   STATUS[967].EXT.AlarmPresent := FALSE;
   STATUS[967].EXT.AlarmFailUnAck := FALSE;
   STATUS[967].Status := 0;
   STATUS[967].TimeStamp := 16#0000;
   STATUS[968].EXT.AlarmWarnUnAck := FALSE;
   STATUS[968].EXT.AckRequired := FALSE;
   STATUS[968].EXT.Maintanence := FALSE;
   STATUS[968].EXT.Operation := FALSE;
   STATUS[968].EXT.Forced := FALSE;
   STATUS[968].EXT.BIT29 := FALSE;
   STATUS[968].EXT.BIT30 := FALSE;
   STATUS[968].EXT.BIT31 := FALSE;
   STATUS[968].EXT.ModeBit1 := FALSE;
   STATUS[968].EXT.ModeBit2 := FALSE;
   STATUS[968].EXT.ModeBit3 := FALSE;
   STATUS[968].EXT.BIT19 := FALSE;
   STATUS[968].EXT.BIT20 := FALSE;
   STATUS[968].EXT.AlarmSuppressed := FALSE;
   STATUS[968].EXT.AlarmPresent := FALSE;
   STATUS[968].EXT.AlarmFailUnAck := FALSE;
   STATUS[968].Status := 0;
   STATUS[968].TimeStamp := 16#0000;
   STATUS[969].EXT.AlarmWarnUnAck := FALSE;
   STATUS[969].EXT.AckRequired := FALSE;
   STATUS[969].EXT.Maintanence := FALSE;
   STATUS[969].EXT.Operation := FALSE;
   STATUS[969].EXT.Forced := FALSE;
   STATUS[969].EXT.BIT29 := FALSE;
   STATUS[969].EXT.BIT30 := FALSE;
   STATUS[969].EXT.BIT31 := FALSE;
   STATUS[969].EXT.ModeBit1 := FALSE;
   STATUS[969].EXT.ModeBit2 := FALSE;
   STATUS[969].EXT.ModeBit3 := FALSE;
   STATUS[969].EXT.BIT19 := FALSE;
   STATUS[969].EXT.BIT20 := FALSE;
   STATUS[969].EXT.AlarmSuppressed := FALSE;
   STATUS[969].EXT.AlarmPresent := FALSE;
   STATUS[969].EXT.AlarmFailUnAck := FALSE;
   STATUS[969].Status := 0;
   STATUS[969].TimeStamp := 16#0000;
   STATUS[970].EXT.AlarmWarnUnAck := FALSE;
   STATUS[970].EXT.AckRequired := FALSE;
   STATUS[970].EXT.Maintanence := FALSE;
   STATUS[970].EXT.Operation := FALSE;
   STATUS[970].EXT.Forced := FALSE;
   STATUS[970].EXT.BIT29 := FALSE;
   STATUS[970].EXT.BIT30 := FALSE;
   STATUS[970].EXT.BIT31 := FALSE;
   STATUS[970].EXT.ModeBit1 := FALSE;
   STATUS[970].EXT.ModeBit2 := FALSE;
   STATUS[970].EXT.ModeBit3 := FALSE;
   STATUS[970].EXT.BIT19 := FALSE;
   STATUS[970].EXT.BIT20 := FALSE;
   STATUS[970].EXT.AlarmSuppressed := FALSE;
   STATUS[970].EXT.AlarmPresent := FALSE;
   STATUS[970].EXT.AlarmFailUnAck := FALSE;
   STATUS[970].Status := 0;
   STATUS[970].TimeStamp := 16#0000;
   STATUS[971].EXT.AlarmWarnUnAck := FALSE;
   STATUS[971].EXT.AckRequired := FALSE;
   STATUS[971].EXT.Maintanence := FALSE;
   STATUS[971].EXT.Operation := FALSE;
   STATUS[971].EXT.Forced := FALSE;
   STATUS[971].EXT.BIT29 := FALSE;
   STATUS[971].EXT.BIT30 := FALSE;
   STATUS[971].EXT.BIT31 := FALSE;
   STATUS[971].EXT.ModeBit1 := FALSE;
   STATUS[971].EXT.ModeBit2 := FALSE;
   STATUS[971].EXT.ModeBit3 := FALSE;
   STATUS[971].EXT.BIT19 := FALSE;
   STATUS[971].EXT.BIT20 := FALSE;
   STATUS[971].EXT.AlarmSuppressed := FALSE;
   STATUS[971].EXT.AlarmPresent := FALSE;
   STATUS[971].EXT.AlarmFailUnAck := FALSE;
   STATUS[971].Status := 0;
   STATUS[971].TimeStamp := 16#0000;
   STATUS[972].EXT.AlarmWarnUnAck := FALSE;
   STATUS[972].EXT.AckRequired := FALSE;
   STATUS[972].EXT.Maintanence := FALSE;
   STATUS[972].EXT.Operation := FALSE;
   STATUS[972].EXT.Forced := FALSE;
   STATUS[972].EXT.BIT29 := FALSE;
   STATUS[972].EXT.BIT30 := FALSE;
   STATUS[972].EXT.BIT31 := FALSE;
   STATUS[972].EXT.ModeBit1 := FALSE;
   STATUS[972].EXT.ModeBit2 := FALSE;
   STATUS[972].EXT.ModeBit3 := FALSE;
   STATUS[972].EXT.BIT19 := FALSE;
   STATUS[972].EXT.BIT20 := FALSE;
   STATUS[972].EXT.AlarmSuppressed := FALSE;
   STATUS[972].EXT.AlarmPresent := FALSE;
   STATUS[972].EXT.AlarmFailUnAck := FALSE;
   STATUS[972].Status := 0;
   STATUS[972].TimeStamp := 16#0000;
   STATUS[973].EXT.AlarmWarnUnAck := FALSE;
   STATUS[973].EXT.AckRequired := FALSE;
   STATUS[973].EXT.Maintanence := FALSE;
   STATUS[973].EXT.Operation := FALSE;
   STATUS[973].EXT.Forced := FALSE;
   STATUS[973].EXT.BIT29 := FALSE;
   STATUS[973].EXT.BIT30 := FALSE;
   STATUS[973].EXT.BIT31 := FALSE;
   STATUS[973].EXT.ModeBit1 := FALSE;
   STATUS[973].EXT.ModeBit2 := FALSE;
   STATUS[973].EXT.ModeBit3 := FALSE;
   STATUS[973].EXT.BIT19 := FALSE;
   STATUS[973].EXT.BIT20 := FALSE;
   STATUS[973].EXT.AlarmSuppressed := FALSE;
   STATUS[973].EXT.AlarmPresent := FALSE;
   STATUS[973].EXT.AlarmFailUnAck := FALSE;
   STATUS[973].Status := 0;
   STATUS[973].TimeStamp := 16#0000;
   STATUS[974].EXT.AlarmWarnUnAck := FALSE;
   STATUS[974].EXT.AckRequired := FALSE;
   STATUS[974].EXT.Maintanence := FALSE;
   STATUS[974].EXT.Operation := FALSE;
   STATUS[974].EXT.Forced := FALSE;
   STATUS[974].EXT.BIT29 := FALSE;
   STATUS[974].EXT.BIT30 := FALSE;
   STATUS[974].EXT.BIT31 := FALSE;
   STATUS[974].EXT.ModeBit1 := FALSE;
   STATUS[974].EXT.ModeBit2 := FALSE;
   STATUS[974].EXT.ModeBit3 := FALSE;
   STATUS[974].EXT.BIT19 := FALSE;
   STATUS[974].EXT.BIT20 := FALSE;
   STATUS[974].EXT.AlarmSuppressed := FALSE;
   STATUS[974].EXT.AlarmPresent := FALSE;
   STATUS[974].EXT.AlarmFailUnAck := FALSE;
   STATUS[974].Status := 0;
   STATUS[974].TimeStamp := 16#0000;
   STATUS[975].EXT.AlarmWarnUnAck := FALSE;
   STATUS[975].EXT.AckRequired := FALSE;
   STATUS[975].EXT.Maintanence := FALSE;
   STATUS[975].EXT.Operation := FALSE;
   STATUS[975].EXT.Forced := FALSE;
   STATUS[975].EXT.BIT29 := FALSE;
   STATUS[975].EXT.BIT30 := FALSE;
   STATUS[975].EXT.BIT31 := FALSE;
   STATUS[975].EXT.ModeBit1 := FALSE;
   STATUS[975].EXT.ModeBit2 := FALSE;
   STATUS[975].EXT.ModeBit3 := FALSE;
   STATUS[975].EXT.BIT19 := FALSE;
   STATUS[975].EXT.BIT20 := FALSE;
   STATUS[975].EXT.AlarmSuppressed := FALSE;
   STATUS[975].EXT.AlarmPresent := FALSE;
   STATUS[975].EXT.AlarmFailUnAck := FALSE;
   STATUS[975].Status := 0;
   STATUS[975].TimeStamp := 16#0000;
   STATUS[976].EXT.AlarmWarnUnAck := FALSE;
   STATUS[976].EXT.AckRequired := FALSE;
   STATUS[976].EXT.Maintanence := FALSE;
   STATUS[976].EXT.Operation := FALSE;
   STATUS[976].EXT.Forced := FALSE;
   STATUS[976].EXT.BIT29 := FALSE;
   STATUS[976].EXT.BIT30 := FALSE;
   STATUS[976].EXT.BIT31 := FALSE;
   STATUS[976].EXT.ModeBit1 := FALSE;
   STATUS[976].EXT.ModeBit2 := FALSE;
   STATUS[976].EXT.ModeBit3 := FALSE;
   STATUS[976].EXT.BIT19 := FALSE;
   STATUS[976].EXT.BIT20 := FALSE;
   STATUS[976].EXT.AlarmSuppressed := FALSE;
   STATUS[976].EXT.AlarmPresent := FALSE;
   STATUS[976].EXT.AlarmFailUnAck := FALSE;
   STATUS[976].Status := 0;
   STATUS[976].TimeStamp := 16#0000;
   STATUS[977].EXT.AlarmWarnUnAck := FALSE;
   STATUS[977].EXT.AckRequired := FALSE;
   STATUS[977].EXT.Maintanence := FALSE;
   STATUS[977].EXT.Operation := FALSE;
   STATUS[977].EXT.Forced := FALSE;
   STATUS[977].EXT.BIT29 := FALSE;
   STATUS[977].EXT.BIT30 := FALSE;
   STATUS[977].EXT.BIT31 := FALSE;
   STATUS[977].EXT.ModeBit1 := FALSE;
   STATUS[977].EXT.ModeBit2 := FALSE;
   STATUS[977].EXT.ModeBit3 := FALSE;
   STATUS[977].EXT.BIT19 := FALSE;
   STATUS[977].EXT.BIT20 := FALSE;
   STATUS[977].EXT.AlarmSuppressed := FALSE;
   STATUS[977].EXT.AlarmPresent := FALSE;
   STATUS[977].EXT.AlarmFailUnAck := FALSE;
   STATUS[977].Status := 0;
   STATUS[977].TimeStamp := 16#0000;
   STATUS[978].EXT.AlarmWarnUnAck := FALSE;
   STATUS[978].EXT.AckRequired := FALSE;
   STATUS[978].EXT.Maintanence := FALSE;
   STATUS[978].EXT.Operation := FALSE;
   STATUS[978].EXT.Forced := FALSE;
   STATUS[978].EXT.BIT29 := FALSE;
   STATUS[978].EXT.BIT30 := FALSE;
   STATUS[978].EXT.BIT31 := FALSE;
   STATUS[978].EXT.ModeBit1 := FALSE;
   STATUS[978].EXT.ModeBit2 := FALSE;
   STATUS[978].EXT.ModeBit3 := FALSE;
   STATUS[978].EXT.BIT19 := FALSE;
   STATUS[978].EXT.BIT20 := FALSE;
   STATUS[978].EXT.AlarmSuppressed := FALSE;
   STATUS[978].EXT.AlarmPresent := FALSE;
   STATUS[978].EXT.AlarmFailUnAck := FALSE;
   STATUS[978].Status := 0;
   STATUS[978].TimeStamp := 16#0000;
   STATUS[979].EXT.AlarmWarnUnAck := FALSE;
   STATUS[979].EXT.AckRequired := FALSE;
   STATUS[979].EXT.Maintanence := FALSE;
   STATUS[979].EXT.Operation := FALSE;
   STATUS[979].EXT.Forced := FALSE;
   STATUS[979].EXT.BIT29 := FALSE;
   STATUS[979].EXT.BIT30 := FALSE;
   STATUS[979].EXT.BIT31 := FALSE;
   STATUS[979].EXT.ModeBit1 := FALSE;
   STATUS[979].EXT.ModeBit2 := FALSE;
   STATUS[979].EXT.ModeBit3 := FALSE;
   STATUS[979].EXT.BIT19 := FALSE;
   STATUS[979].EXT.BIT20 := FALSE;
   STATUS[979].EXT.AlarmSuppressed := FALSE;
   STATUS[979].EXT.AlarmPresent := FALSE;
   STATUS[979].EXT.AlarmFailUnAck := FALSE;
   STATUS[979].Status := 0;
   STATUS[979].TimeStamp := 16#0000;
   STATUS[980].EXT.AlarmWarnUnAck := FALSE;
   STATUS[980].EXT.AckRequired := FALSE;
   STATUS[980].EXT.Maintanence := FALSE;
   STATUS[980].EXT.Operation := FALSE;
   STATUS[980].EXT.Forced := FALSE;
   STATUS[980].EXT.BIT29 := FALSE;
   STATUS[980].EXT.BIT30 := FALSE;
   STATUS[980].EXT.BIT31 := FALSE;
   STATUS[980].EXT.ModeBit1 := FALSE;
   STATUS[980].EXT.ModeBit2 := FALSE;
   STATUS[980].EXT.ModeBit3 := FALSE;
   STATUS[980].EXT.BIT19 := FALSE;
   STATUS[980].EXT.BIT20 := FALSE;
   STATUS[980].EXT.AlarmSuppressed := FALSE;
   STATUS[980].EXT.AlarmPresent := FALSE;
   STATUS[980].EXT.AlarmFailUnAck := FALSE;
   STATUS[980].Status := 0;
   STATUS[980].TimeStamp := 16#0000;
   STATUS[981].EXT.AlarmWarnUnAck := FALSE;
   STATUS[981].EXT.AckRequired := FALSE;
   STATUS[981].EXT.Maintanence := FALSE;
   STATUS[981].EXT.Operation := FALSE;
   STATUS[981].EXT.Forced := FALSE;
   STATUS[981].EXT.BIT29 := FALSE;
   STATUS[981].EXT.BIT30 := FALSE;
   STATUS[981].EXT.BIT31 := FALSE;
   STATUS[981].EXT.ModeBit1 := FALSE;
   STATUS[981].EXT.ModeBit2 := FALSE;
   STATUS[981].EXT.ModeBit3 := FALSE;
   STATUS[981].EXT.BIT19 := FALSE;
   STATUS[981].EXT.BIT20 := FALSE;
   STATUS[981].EXT.AlarmSuppressed := FALSE;
   STATUS[981].EXT.AlarmPresent := FALSE;
   STATUS[981].EXT.AlarmFailUnAck := FALSE;
   STATUS[981].Status := 0;
   STATUS[981].TimeStamp := 16#0000;
   STATUS[982].EXT.AlarmWarnUnAck := FALSE;
   STATUS[982].EXT.AckRequired := FALSE;
   STATUS[982].EXT.Maintanence := FALSE;
   STATUS[982].EXT.Operation := FALSE;
   STATUS[982].EXT.Forced := FALSE;
   STATUS[982].EXT.BIT29 := FALSE;
   STATUS[982].EXT.BIT30 := FALSE;
   STATUS[982].EXT.BIT31 := FALSE;
   STATUS[982].EXT.ModeBit1 := FALSE;
   STATUS[982].EXT.ModeBit2 := FALSE;
   STATUS[982].EXT.ModeBit3 := FALSE;
   STATUS[982].EXT.BIT19 := FALSE;
   STATUS[982].EXT.BIT20 := FALSE;
   STATUS[982].EXT.AlarmSuppressed := FALSE;
   STATUS[982].EXT.AlarmPresent := FALSE;
   STATUS[982].EXT.AlarmFailUnAck := FALSE;
   STATUS[982].Status := 0;
   STATUS[982].TimeStamp := 16#0000;
   STATUS[983].EXT.AlarmWarnUnAck := FALSE;
   STATUS[983].EXT.AckRequired := FALSE;
   STATUS[983].EXT.Maintanence := FALSE;
   STATUS[983].EXT.Operation := FALSE;
   STATUS[983].EXT.Forced := FALSE;
   STATUS[983].EXT.BIT29 := FALSE;
   STATUS[983].EXT.BIT30 := FALSE;
   STATUS[983].EXT.BIT31 := FALSE;
   STATUS[983].EXT.ModeBit1 := FALSE;
   STATUS[983].EXT.ModeBit2 := FALSE;
   STATUS[983].EXT.ModeBit3 := FALSE;
   STATUS[983].EXT.BIT19 := FALSE;
   STATUS[983].EXT.BIT20 := FALSE;
   STATUS[983].EXT.AlarmSuppressed := FALSE;
   STATUS[983].EXT.AlarmPresent := FALSE;
   STATUS[983].EXT.AlarmFailUnAck := FALSE;
   STATUS[983].Status := 0;
   STATUS[983].TimeStamp := 16#0000;
   STATUS[984].EXT.AlarmWarnUnAck := FALSE;
   STATUS[984].EXT.AckRequired := FALSE;
   STATUS[984].EXT.Maintanence := FALSE;
   STATUS[984].EXT.Operation := FALSE;
   STATUS[984].EXT.Forced := FALSE;
   STATUS[984].EXT.BIT29 := FALSE;
   STATUS[984].EXT.BIT30 := FALSE;
   STATUS[984].EXT.BIT31 := FALSE;
   STATUS[984].EXT.ModeBit1 := FALSE;
   STATUS[984].EXT.ModeBit2 := FALSE;
   STATUS[984].EXT.ModeBit3 := FALSE;
   STATUS[984].EXT.BIT19 := FALSE;
   STATUS[984].EXT.BIT20 := FALSE;
   STATUS[984].EXT.AlarmSuppressed := FALSE;
   STATUS[984].EXT.AlarmPresent := FALSE;
   STATUS[984].EXT.AlarmFailUnAck := FALSE;
   STATUS[984].Status := 0;
   STATUS[984].TimeStamp := 16#0000;
   STATUS[985].EXT.AlarmWarnUnAck := FALSE;
   STATUS[985].EXT.AckRequired := FALSE;
   STATUS[985].EXT.Maintanence := FALSE;
   STATUS[985].EXT.Operation := FALSE;
   STATUS[985].EXT.Forced := FALSE;
   STATUS[985].EXT.BIT29 := FALSE;
   STATUS[985].EXT.BIT30 := FALSE;
   STATUS[985].EXT.BIT31 := FALSE;
   STATUS[985].EXT.ModeBit1 := FALSE;
   STATUS[985].EXT.ModeBit2 := FALSE;
   STATUS[985].EXT.ModeBit3 := FALSE;
   STATUS[985].EXT.BIT19 := FALSE;
   STATUS[985].EXT.BIT20 := FALSE;
   STATUS[985].EXT.AlarmSuppressed := FALSE;
   STATUS[985].EXT.AlarmPresent := FALSE;
   STATUS[985].EXT.AlarmFailUnAck := FALSE;
   STATUS[985].Status := 0;
   STATUS[985].TimeStamp := 16#0000;
   STATUS[986].EXT.AlarmWarnUnAck := FALSE;
   STATUS[986].EXT.AckRequired := FALSE;
   STATUS[986].EXT.Maintanence := FALSE;
   STATUS[986].EXT.Operation := FALSE;
   STATUS[986].EXT.Forced := FALSE;
   STATUS[986].EXT.BIT29 := FALSE;
   STATUS[986].EXT.BIT30 := FALSE;
   STATUS[986].EXT.BIT31 := FALSE;
   STATUS[986].EXT.ModeBit1 := FALSE;
   STATUS[986].EXT.ModeBit2 := FALSE;
   STATUS[986].EXT.ModeBit3 := FALSE;
   STATUS[986].EXT.BIT19 := FALSE;
   STATUS[986].EXT.BIT20 := FALSE;
   STATUS[986].EXT.AlarmSuppressed := FALSE;
   STATUS[986].EXT.AlarmPresent := FALSE;
   STATUS[986].EXT.AlarmFailUnAck := FALSE;
   STATUS[986].Status := 0;
   STATUS[986].TimeStamp := 16#0000;
   STATUS[987].EXT.AlarmWarnUnAck := FALSE;
   STATUS[987].EXT.AckRequired := FALSE;
   STATUS[987].EXT.Maintanence := FALSE;
   STATUS[987].EXT.Operation := FALSE;
   STATUS[987].EXT.Forced := FALSE;
   STATUS[987].EXT.BIT29 := FALSE;
   STATUS[987].EXT.BIT30 := FALSE;
   STATUS[987].EXT.BIT31 := FALSE;
   STATUS[987].EXT.ModeBit1 := FALSE;
   STATUS[987].EXT.ModeBit2 := FALSE;
   STATUS[987].EXT.ModeBit3 := FALSE;
   STATUS[987].EXT.BIT19 := FALSE;
   STATUS[987].EXT.BIT20 := FALSE;
   STATUS[987].EXT.AlarmSuppressed := FALSE;
   STATUS[987].EXT.AlarmPresent := FALSE;
   STATUS[987].EXT.AlarmFailUnAck := FALSE;
   STATUS[987].Status := 0;
   STATUS[987].TimeStamp := 16#0000;
   STATUS[988].EXT.AlarmWarnUnAck := FALSE;
   STATUS[988].EXT.AckRequired := FALSE;
   STATUS[988].EXT.Maintanence := FALSE;
   STATUS[988].EXT.Operation := FALSE;
   STATUS[988].EXT.Forced := FALSE;
   STATUS[988].EXT.BIT29 := FALSE;
   STATUS[988].EXT.BIT30 := FALSE;
   STATUS[988].EXT.BIT31 := FALSE;
   STATUS[988].EXT.ModeBit1 := FALSE;
   STATUS[988].EXT.ModeBit2 := FALSE;
   STATUS[988].EXT.ModeBit3 := FALSE;
   STATUS[988].EXT.BIT19 := FALSE;
   STATUS[988].EXT.BIT20 := FALSE;
   STATUS[988].EXT.AlarmSuppressed := FALSE;
   STATUS[988].EXT.AlarmPresent := FALSE;
   STATUS[988].EXT.AlarmFailUnAck := FALSE;
   STATUS[988].Status := 0;
   STATUS[988].TimeStamp := 16#0000;
   STATUS[989].EXT.AlarmWarnUnAck := FALSE;
   STATUS[989].EXT.AckRequired := FALSE;
   STATUS[989].EXT.Maintanence := FALSE;
   STATUS[989].EXT.Operation := FALSE;
   STATUS[989].EXT.Forced := FALSE;
   STATUS[989].EXT.BIT29 := FALSE;
   STATUS[989].EXT.BIT30 := FALSE;
   STATUS[989].EXT.BIT31 := FALSE;
   STATUS[989].EXT.ModeBit1 := FALSE;
   STATUS[989].EXT.ModeBit2 := FALSE;
   STATUS[989].EXT.ModeBit3 := FALSE;
   STATUS[989].EXT.BIT19 := FALSE;
   STATUS[989].EXT.BIT20 := FALSE;
   STATUS[989].EXT.AlarmSuppressed := FALSE;
   STATUS[989].EXT.AlarmPresent := FALSE;
   STATUS[989].EXT.AlarmFailUnAck := FALSE;
   STATUS[989].Status := 0;
   STATUS[989].TimeStamp := 16#0000;
   STATUS[990].EXT.AlarmWarnUnAck := FALSE;
   STATUS[990].EXT.AckRequired := FALSE;
   STATUS[990].EXT.Maintanence := FALSE;
   STATUS[990].EXT.Operation := FALSE;
   STATUS[990].EXT.Forced := FALSE;
   STATUS[990].EXT.BIT29 := FALSE;
   STATUS[990].EXT.BIT30 := FALSE;
   STATUS[990].EXT.BIT31 := FALSE;
   STATUS[990].EXT.ModeBit1 := FALSE;
   STATUS[990].EXT.ModeBit2 := FALSE;
   STATUS[990].EXT.ModeBit3 := FALSE;
   STATUS[990].EXT.BIT19 := FALSE;
   STATUS[990].EXT.BIT20 := FALSE;
   STATUS[990].EXT.AlarmSuppressed := FALSE;
   STATUS[990].EXT.AlarmPresent := FALSE;
   STATUS[990].EXT.AlarmFailUnAck := FALSE;
   STATUS[990].Status := 0;
   STATUS[990].TimeStamp := 16#0000;
   STATUS[991].EXT.AlarmWarnUnAck := FALSE;
   STATUS[991].EXT.AckRequired := FALSE;
   STATUS[991].EXT.Maintanence := FALSE;
   STATUS[991].EXT.Operation := FALSE;
   STATUS[991].EXT.Forced := FALSE;
   STATUS[991].EXT.BIT29 := FALSE;
   STATUS[991].EXT.BIT30 := FALSE;
   STATUS[991].EXT.BIT31 := FALSE;
   STATUS[991].EXT.ModeBit1 := FALSE;
   STATUS[991].EXT.ModeBit2 := FALSE;
   STATUS[991].EXT.ModeBit3 := FALSE;
   STATUS[991].EXT.BIT19 := FALSE;
   STATUS[991].EXT.BIT20 := FALSE;
   STATUS[991].EXT.AlarmSuppressed := FALSE;
   STATUS[991].EXT.AlarmPresent := FALSE;
   STATUS[991].EXT.AlarmFailUnAck := FALSE;
   STATUS[991].Status := 0;
   STATUS[991].TimeStamp := 16#0000;
   STATUS[992].EXT.AlarmWarnUnAck := FALSE;
   STATUS[992].EXT.AckRequired := FALSE;
   STATUS[992].EXT.Maintanence := FALSE;
   STATUS[992].EXT.Operation := FALSE;
   STATUS[992].EXT.Forced := FALSE;
   STATUS[992].EXT.BIT29 := FALSE;
   STATUS[992].EXT.BIT30 := FALSE;
   STATUS[992].EXT.BIT31 := FALSE;
   STATUS[992].EXT.ModeBit1 := FALSE;
   STATUS[992].EXT.ModeBit2 := FALSE;
   STATUS[992].EXT.ModeBit3 := FALSE;
   STATUS[992].EXT.BIT19 := FALSE;
   STATUS[992].EXT.BIT20 := FALSE;
   STATUS[992].EXT.AlarmSuppressed := FALSE;
   STATUS[992].EXT.AlarmPresent := FALSE;
   STATUS[992].EXT.AlarmFailUnAck := FALSE;
   STATUS[992].Status := 0;
   STATUS[992].TimeStamp := 16#0000;
   STATUS[993].EXT.AlarmWarnUnAck := FALSE;
   STATUS[993].EXT.AckRequired := FALSE;
   STATUS[993].EXT.Maintanence := FALSE;
   STATUS[993].EXT.Operation := FALSE;
   STATUS[993].EXT.Forced := FALSE;
   STATUS[993].EXT.BIT29 := FALSE;
   STATUS[993].EXT.BIT30 := FALSE;
   STATUS[993].EXT.BIT31 := FALSE;
   STATUS[993].EXT.ModeBit1 := FALSE;
   STATUS[993].EXT.ModeBit2 := FALSE;
   STATUS[993].EXT.ModeBit3 := FALSE;
   STATUS[993].EXT.BIT19 := FALSE;
   STATUS[993].EXT.BIT20 := FALSE;
   STATUS[993].EXT.AlarmSuppressed := FALSE;
   STATUS[993].EXT.AlarmPresent := FALSE;
   STATUS[993].EXT.AlarmFailUnAck := FALSE;
   STATUS[993].Status := 0;
   STATUS[993].TimeStamp := 16#0000;
   STATUS[994].EXT.AlarmWarnUnAck := FALSE;
   STATUS[994].EXT.AckRequired := FALSE;
   STATUS[994].EXT.Maintanence := FALSE;
   STATUS[994].EXT.Operation := FALSE;
   STATUS[994].EXT.Forced := FALSE;
   STATUS[994].EXT.BIT29 := FALSE;
   STATUS[994].EXT.BIT30 := FALSE;
   STATUS[994].EXT.BIT31 := FALSE;
   STATUS[994].EXT.ModeBit1 := FALSE;
   STATUS[994].EXT.ModeBit2 := FALSE;
   STATUS[994].EXT.ModeBit3 := FALSE;
   STATUS[994].EXT.BIT19 := FALSE;
   STATUS[994].EXT.BIT20 := FALSE;
   STATUS[994].EXT.AlarmSuppressed := FALSE;
   STATUS[994].EXT.AlarmPresent := FALSE;
   STATUS[994].EXT.AlarmFailUnAck := FALSE;
   STATUS[994].Status := 0;
   STATUS[994].TimeStamp := 16#0000;
   STATUS[995].EXT.AlarmWarnUnAck := FALSE;
   STATUS[995].EXT.AckRequired := FALSE;
   STATUS[995].EXT.Maintanence := FALSE;
   STATUS[995].EXT.Operation := FALSE;
   STATUS[995].EXT.Forced := FALSE;
   STATUS[995].EXT.BIT29 := FALSE;
   STATUS[995].EXT.BIT30 := FALSE;
   STATUS[995].EXT.BIT31 := FALSE;
   STATUS[995].EXT.ModeBit1 := FALSE;
   STATUS[995].EXT.ModeBit2 := FALSE;
   STATUS[995].EXT.ModeBit3 := FALSE;
   STATUS[995].EXT.BIT19 := FALSE;
   STATUS[995].EXT.BIT20 := FALSE;
   STATUS[995].EXT.AlarmSuppressed := FALSE;
   STATUS[995].EXT.AlarmPresent := FALSE;
   STATUS[995].EXT.AlarmFailUnAck := FALSE;
   STATUS[995].Status := 0;
   STATUS[995].TimeStamp := 16#0000;
   STATUS[996].EXT.AlarmWarnUnAck := FALSE;
   STATUS[996].EXT.AckRequired := FALSE;
   STATUS[996].EXT.Maintanence := FALSE;
   STATUS[996].EXT.Operation := FALSE;
   STATUS[996].EXT.Forced := FALSE;
   STATUS[996].EXT.BIT29 := FALSE;
   STATUS[996].EXT.BIT30 := FALSE;
   STATUS[996].EXT.BIT31 := FALSE;
   STATUS[996].EXT.ModeBit1 := FALSE;
   STATUS[996].EXT.ModeBit2 := FALSE;
   STATUS[996].EXT.ModeBit3 := FALSE;
   STATUS[996].EXT.BIT19 := FALSE;
   STATUS[996].EXT.BIT20 := FALSE;
   STATUS[996].EXT.AlarmSuppressed := FALSE;
   STATUS[996].EXT.AlarmPresent := FALSE;
   STATUS[996].EXT.AlarmFailUnAck := FALSE;
   STATUS[996].Status := 0;
   STATUS[996].TimeStamp := 16#0000;
   STATUS[997].EXT.AlarmWarnUnAck := FALSE;
   STATUS[997].EXT.AckRequired := FALSE;
   STATUS[997].EXT.Maintanence := FALSE;
   STATUS[997].EXT.Operation := FALSE;
   STATUS[997].EXT.Forced := FALSE;
   STATUS[997].EXT.BIT29 := FALSE;
   STATUS[997].EXT.BIT30 := FALSE;
   STATUS[997].EXT.BIT31 := FALSE;
   STATUS[997].EXT.ModeBit1 := FALSE;
   STATUS[997].EXT.ModeBit2 := FALSE;
   STATUS[997].EXT.ModeBit3 := FALSE;
   STATUS[997].EXT.BIT19 := FALSE;
   STATUS[997].EXT.BIT20 := FALSE;
   STATUS[997].EXT.AlarmSuppressed := FALSE;
   STATUS[997].EXT.AlarmPresent := FALSE;
   STATUS[997].EXT.AlarmFailUnAck := FALSE;
   STATUS[997].Status := 0;
   STATUS[997].TimeStamp := 16#0000;
   STATUS[998].EXT.AlarmWarnUnAck := FALSE;
   STATUS[998].EXT.AckRequired := FALSE;
   STATUS[998].EXT.Maintanence := FALSE;
   STATUS[998].EXT.Operation := FALSE;
   STATUS[998].EXT.Forced := FALSE;
   STATUS[998].EXT.BIT29 := FALSE;
   STATUS[998].EXT.BIT30 := FALSE;
   STATUS[998].EXT.BIT31 := FALSE;
   STATUS[998].EXT.ModeBit1 := FALSE;
   STATUS[998].EXT.ModeBit2 := FALSE;
   STATUS[998].EXT.ModeBit3 := FALSE;
   STATUS[998].EXT.BIT19 := FALSE;
   STATUS[998].EXT.BIT20 := FALSE;
   STATUS[998].EXT.AlarmSuppressed := FALSE;
   STATUS[998].EXT.AlarmPresent := FALSE;
   STATUS[998].EXT.AlarmFailUnAck := FALSE;
   STATUS[998].Status := 0;
   STATUS[998].TimeStamp := 16#0000;
   STATUS[999].EXT.AlarmWarnUnAck := FALSE;
   STATUS[999].EXT.AckRequired := FALSE;
   STATUS[999].EXT.Maintanence := FALSE;
   STATUS[999].EXT.Operation := FALSE;
   STATUS[999].EXT.Forced := FALSE;
   STATUS[999].EXT.BIT29 := FALSE;
   STATUS[999].EXT.BIT30 := FALSE;
   STATUS[999].EXT.BIT31 := FALSE;
   STATUS[999].EXT.ModeBit1 := FALSE;
   STATUS[999].EXT.ModeBit2 := FALSE;
   STATUS[999].EXT.ModeBit3 := FALSE;
   STATUS[999].EXT.BIT19 := FALSE;
   STATUS[999].EXT.BIT20 := FALSE;
   STATUS[999].EXT.AlarmSuppressed := FALSE;
   STATUS[999].EXT.AlarmPresent := FALSE;
   STATUS[999].EXT.AlarmFailUnAck := FALSE;
   STATUS[999].Status := 0;
   STATUS[999].TimeStamp := 16#0000;
   STATUS[1000].EXT.AlarmWarnUnAck := FALSE;
   STATUS[1000].EXT.AckRequired := FALSE;
   STATUS[1000].EXT.Maintanence := FALSE;
   STATUS[1000].EXT.Operation := FALSE;
   STATUS[1000].EXT.Forced := FALSE;
   STATUS[1000].EXT.BIT29 := FALSE;
   STATUS[1000].EXT.BIT30 := FALSE;
   STATUS[1000].EXT.BIT31 := FALSE;
   STATUS[1000].EXT.ModeBit1 := FALSE;
   STATUS[1000].EXT.ModeBit2 := FALSE;
   STATUS[1000].EXT.ModeBit3 := FALSE;
   STATUS[1000].EXT.BIT19 := FALSE;
   STATUS[1000].EXT.BIT20 := FALSE;
   STATUS[1000].EXT.AlarmSuppressed := FALSE;
   STATUS[1000].EXT.AlarmPresent := FALSE;
   STATUS[1000].EXT.AlarmFailUnAck := FALSE;
   STATUS[1000].Status := 0;
   STATUS[1000].TimeStamp := 16#0000;
END_DATA_BLOCK

DATA_BLOCK "ACESYS_HMI_ANALOG"   // DB7
TITLE = ACESYS ANALOG DB
{ S7_Optimized_Access := 'FALSE' }
AUTHOR : METIS
FAMILY : ACESYS
NAME : AnalogDB
VERSION : 8.0
   VAR
      STATUS : Array[0..1000] of "ACESYS_HMI_STAT_ANALOG";   // Analog Status to HMI
   END_VAR
BEGIN
   STATUS[0].VALUE := 0.0;
   STATUS[0].TRIGVALUE := 0.0;
   STATUS[0].EXT.AlarmWarnUnAck := FALSE;
   STATUS[0].EXT.AckRequired := FALSE;
   STATUS[0].EXT.Maintanence := FALSE;
   STATUS[0].EXT.Operation := FALSE;
   STATUS[0].EXT.Forced := FALSE;
   STATUS[0].EXT.BIT29 := FALSE;
   STATUS[0].EXT.BIT30 := FALSE;
   STATUS[0].EXT.BIT31 := FALSE;
   STATUS[0].EXT.ModeBit1 := FALSE;
   STATUS[0].EXT.ModeBit2 := FALSE;
   STATUS[0].EXT.ModeBit3 := FALSE;
   STATUS[0].EXT.BIT19 := FALSE;
   STATUS[0].EXT.BIT20 := FALSE;
   STATUS[0].EXT.AlarmSuppressed := FALSE;
   STATUS[0].EXT.AlarmPrsent := FALSE;
   STATUS[0].EXT.AlarmFailUnAck := FALSE;
   STATUS[0].Status := 0;
   STATUS[0].TimeStamp := 16#0000;
   STATUS[1].VALUE := 26.11762;
   STATUS[1].TRIGVALUE := 0.0;
   STATUS[1].EXT.AlarmWarnUnAck := TRUE;
   STATUS[1].EXT.AckRequired := FALSE;
   STATUS[1].EXT.Maintanence := FALSE;
   STATUS[1].EXT.Operation := TRUE;
   STATUS[1].EXT.Forced := FALSE;
   STATUS[1].EXT.BIT29 := FALSE;
   STATUS[1].EXT.BIT30 := FALSE;
   STATUS[1].EXT.BIT31 := FALSE;
   STATUS[1].EXT.ModeBit1 := FALSE;
   STATUS[1].EXT.ModeBit2 := FALSE;
   STATUS[1].EXT.ModeBit3 := FALSE;
   STATUS[1].EXT.BIT19 := FALSE;
   STATUS[1].EXT.BIT20 := FALSE;
   STATUS[1].EXT.AlarmSuppressed := TRUE;
   STATUS[1].EXT.AlarmPrsent := FALSE;
   STATUS[1].EXT.AlarmFailUnAck := FALSE;
   STATUS[1].Status := 1;
   STATUS[1].TimeStamp := 16#70C1;
   STATUS[2].VALUE := 0.0;
   STATUS[2].TRIGVALUE := 207.17;
   STATUS[2].EXT.AlarmWarnUnAck := TRUE;
   STATUS[2].EXT.AckRequired := FALSE;
   STATUS[2].EXT.Maintanence := FALSE;
   STATUS[2].EXT.Operation := TRUE;
   STATUS[2].EXT.Forced := FALSE;
   STATUS[2].EXT.BIT29 := FALSE;
   STATUS[2].EXT.BIT30 := FALSE;
   STATUS[2].EXT.BIT31 := FALSE;
   STATUS[2].EXT.ModeBit1 := FALSE;
   STATUS[2].EXT.ModeBit2 := FALSE;
   STATUS[2].EXT.ModeBit3 := FALSE;
   STATUS[2].EXT.BIT19 := FALSE;
   STATUS[2].EXT.BIT20 := FALSE;
   STATUS[2].EXT.AlarmSuppressed := FALSE;
   STATUS[2].EXT.AlarmPrsent := FALSE;
   STATUS[2].EXT.AlarmFailUnAck := FALSE;
   STATUS[2].Status := 1;
   STATUS[2].TimeStamp := 16#1C48;
   STATUS[3].VALUE := 0.0;
   STATUS[3].TRIGVALUE := 0.0;
   STATUS[3].EXT.AlarmWarnUnAck := TRUE;
   STATUS[3].EXT.AckRequired := FALSE;
   STATUS[3].EXT.Maintanence := FALSE;
   STATUS[3].EXT.Operation := TRUE;
   STATUS[3].EXT.Forced := FALSE;
   STATUS[3].EXT.BIT29 := FALSE;
   STATUS[3].EXT.BIT30 := FALSE;
   STATUS[3].EXT.BIT31 := FALSE;
   STATUS[3].EXT.ModeBit1 := FALSE;
   STATUS[3].EXT.ModeBit2 := FALSE;
   STATUS[3].EXT.ModeBit3 := FALSE;
   STATUS[3].EXT.BIT19 := FALSE;
   STATUS[3].EXT.BIT20 := FALSE;
   STATUS[3].EXT.AlarmSuppressed := TRUE;
   STATUS[3].EXT.AlarmPrsent := FALSE;
   STATUS[3].EXT.AlarmFailUnAck := FALSE;
   STATUS[3].Status := 1;
   STATUS[3].TimeStamp := 16#3928;
   STATUS[4].VALUE := 0.0;
   STATUS[4].TRIGVALUE := 0.0;
   STATUS[4].EXT.AlarmWarnUnAck := TRUE;
   STATUS[4].EXT.AckRequired := FALSE;
   STATUS[4].EXT.Maintanence := FALSE;
   STATUS[4].EXT.Operation := TRUE;
   STATUS[4].EXT.Forced := FALSE;
   STATUS[4].EXT.BIT29 := FALSE;
   STATUS[4].EXT.BIT30 := FALSE;
   STATUS[4].EXT.BIT31 := FALSE;
   STATUS[4].EXT.ModeBit1 := FALSE;
   STATUS[4].EXT.ModeBit2 := FALSE;
   STATUS[4].EXT.ModeBit3 := FALSE;
   STATUS[4].EXT.BIT19 := FALSE;
   STATUS[4].EXT.BIT20 := FALSE;
   STATUS[4].EXT.AlarmSuppressed := TRUE;
   STATUS[4].EXT.AlarmPrsent := FALSE;
   STATUS[4].EXT.AlarmFailUnAck := FALSE;
   STATUS[4].Status := 1;
   STATUS[4].TimeStamp := 16#3928;
   STATUS[5].VALUE := 0.0;
   STATUS[5].TRIGVALUE := 0.0;
   STATUS[5].EXT.AlarmWarnUnAck := TRUE;
   STATUS[5].EXT.AckRequired := FALSE;
   STATUS[5].EXT.Maintanence := FALSE;
   STATUS[5].EXT.Operation := TRUE;
   STATUS[5].EXT.Forced := FALSE;
   STATUS[5].EXT.BIT29 := FALSE;
   STATUS[5].EXT.BIT30 := FALSE;
   STATUS[5].EXT.BIT31 := FALSE;
   STATUS[5].EXT.ModeBit1 := FALSE;
   STATUS[5].EXT.ModeBit2 := FALSE;
   STATUS[5].EXT.ModeBit3 := FALSE;
   STATUS[5].EXT.BIT19 := FALSE;
   STATUS[5].EXT.BIT20 := FALSE;
   STATUS[5].EXT.AlarmSuppressed := FALSE;
   STATUS[5].EXT.AlarmPrsent := FALSE;
   STATUS[5].EXT.AlarmFailUnAck := FALSE;
   STATUS[5].Status := 1;
   STATUS[5].TimeStamp := 16#B1BD;
   STATUS[6].VALUE := 0.0;
   STATUS[6].TRIGVALUE := 0.0;
   STATUS[6].EXT.AlarmWarnUnAck := TRUE;
   STATUS[6].EXT.AckRequired := FALSE;
   STATUS[6].EXT.Maintanence := FALSE;
   STATUS[6].EXT.Operation := TRUE;
   STATUS[6].EXT.Forced := FALSE;
   STATUS[6].EXT.BIT29 := FALSE;
   STATUS[6].EXT.BIT30 := FALSE;
   STATUS[6].EXT.BIT31 := FALSE;
   STATUS[6].EXT.ModeBit1 := FALSE;
   STATUS[6].EXT.ModeBit2 := FALSE;
   STATUS[6].EXT.ModeBit3 := FALSE;
   STATUS[6].EXT.BIT19 := FALSE;
   STATUS[6].EXT.BIT20 := FALSE;
   STATUS[6].EXT.AlarmSuppressed := FALSE;
   STATUS[6].EXT.AlarmPrsent := FALSE;
   STATUS[6].EXT.AlarmFailUnAck := FALSE;
   STATUS[6].Status := 1;
   STATUS[6].TimeStamp := 16#9BAA;
   STATUS[7].VALUE := 0.0;
   STATUS[7].TRIGVALUE := 0.0;
   STATUS[7].EXT.AlarmWarnUnAck := TRUE;
   STATUS[7].EXT.AckRequired := FALSE;
   STATUS[7].EXT.Maintanence := FALSE;
   STATUS[7].EXT.Operation := TRUE;
   STATUS[7].EXT.Forced := FALSE;
   STATUS[7].EXT.BIT29 := FALSE;
   STATUS[7].EXT.BIT30 := FALSE;
   STATUS[7].EXT.BIT31 := FALSE;
   STATUS[7].EXT.ModeBit1 := FALSE;
   STATUS[7].EXT.ModeBit2 := FALSE;
   STATUS[7].EXT.ModeBit3 := FALSE;
   STATUS[7].EXT.BIT19 := FALSE;
   STATUS[7].EXT.BIT20 := FALSE;
   STATUS[7].EXT.AlarmSuppressed := TRUE;
   STATUS[7].EXT.AlarmPrsent := FALSE;
   STATUS[7].EXT.AlarmFailUnAck := FALSE;
   STATUS[7].Status := 1;
   STATUS[7].TimeStamp := 16#3928;
   STATUS[8].VALUE := 0.0;
   STATUS[8].TRIGVALUE := 90.0;
   STATUS[8].EXT.AlarmWarnUnAck := TRUE;
   STATUS[8].EXT.AckRequired := FALSE;
   STATUS[8].EXT.Maintanence := FALSE;
   STATUS[8].EXT.Operation := TRUE;
   STATUS[8].EXT.Forced := FALSE;
   STATUS[8].EXT.BIT29 := FALSE;
   STATUS[8].EXT.BIT30 := FALSE;
   STATUS[8].EXT.BIT31 := FALSE;
   STATUS[8].EXT.ModeBit1 := FALSE;
   STATUS[8].EXT.ModeBit2 := FALSE;
   STATUS[8].EXT.ModeBit3 := FALSE;
   STATUS[8].EXT.BIT19 := FALSE;
   STATUS[8].EXT.BIT20 := FALSE;
   STATUS[8].EXT.AlarmSuppressed := TRUE;
   STATUS[8].EXT.AlarmPrsent := FALSE;
   STATUS[8].EXT.AlarmFailUnAck := FALSE;
   STATUS[8].Status := 1;
   STATUS[8].TimeStamp := 16#399B;
   STATUS[9].VALUE := 0.0;
   STATUS[9].TRIGVALUE := 0.0;
   STATUS[9].EXT.AlarmWarnUnAck := TRUE;
   STATUS[9].EXT.AckRequired := FALSE;
   STATUS[9].EXT.Maintanence := FALSE;
   STATUS[9].EXT.Operation := TRUE;
   STATUS[9].EXT.Forced := FALSE;
   STATUS[9].EXT.BIT29 := FALSE;
   STATUS[9].EXT.BIT30 := FALSE;
   STATUS[9].EXT.BIT31 := FALSE;
   STATUS[9].EXT.ModeBit1 := FALSE;
   STATUS[9].EXT.ModeBit2 := FALSE;
   STATUS[9].EXT.ModeBit3 := FALSE;
   STATUS[9].EXT.BIT19 := FALSE;
   STATUS[9].EXT.BIT20 := FALSE;
   STATUS[9].EXT.AlarmSuppressed := FALSE;
   STATUS[9].EXT.AlarmPrsent := FALSE;
   STATUS[9].EXT.AlarmFailUnAck := FALSE;
   STATUS[9].Status := 1;
   STATUS[9].TimeStamp := 16#3928;
   STATUS[10].VALUE := 0.0;
   STATUS[10].TRIGVALUE := 0.0;
   STATUS[10].EXT.AlarmWarnUnAck := TRUE;
   STATUS[10].EXT.AckRequired := FALSE;
   STATUS[10].EXT.Maintanence := FALSE;
   STATUS[10].EXT.Operation := TRUE;
   STATUS[10].EXT.Forced := FALSE;
   STATUS[10].EXT.BIT29 := FALSE;
   STATUS[10].EXT.BIT30 := FALSE;
   STATUS[10].EXT.BIT31 := FALSE;
   STATUS[10].EXT.ModeBit1 := FALSE;
   STATUS[10].EXT.ModeBit2 := FALSE;
   STATUS[10].EXT.ModeBit3 := FALSE;
   STATUS[10].EXT.BIT19 := FALSE;
   STATUS[10].EXT.BIT20 := FALSE;
   STATUS[10].EXT.AlarmSuppressed := FALSE;
   STATUS[10].EXT.AlarmPrsent := FALSE;
   STATUS[10].EXT.AlarmFailUnAck := FALSE;
   STATUS[10].Status := 1;
   STATUS[10].TimeStamp := 16#3928;
   STATUS[11].VALUE := 0.0;
   STATUS[11].TRIGVALUE := 0.0;
   STATUS[11].EXT.AlarmWarnUnAck := TRUE;
   STATUS[11].EXT.AckRequired := FALSE;
   STATUS[11].EXT.Maintanence := FALSE;
   STATUS[11].EXT.Operation := TRUE;
   STATUS[11].EXT.Forced := FALSE;
   STATUS[11].EXT.BIT29 := FALSE;
   STATUS[11].EXT.BIT30 := FALSE;
   STATUS[11].EXT.BIT31 := FALSE;
   STATUS[11].EXT.ModeBit1 := FALSE;
   STATUS[11].EXT.ModeBit2 := FALSE;
   STATUS[11].EXT.ModeBit3 := FALSE;
   STATUS[11].EXT.BIT19 := FALSE;
   STATUS[11].EXT.BIT20 := FALSE;
   STATUS[11].EXT.AlarmSuppressed := TRUE;
   STATUS[11].EXT.AlarmPrsent := FALSE;
   STATUS[11].EXT.AlarmFailUnAck := FALSE;
   STATUS[11].Status := 1;
   STATUS[11].TimeStamp := 16#3928;
   STATUS[12].VALUE := 0.0;
   STATUS[12].TRIGVALUE := 0.0;
   STATUS[12].EXT.AlarmWarnUnAck := TRUE;
   STATUS[12].EXT.AckRequired := FALSE;
   STATUS[12].EXT.Maintanence := FALSE;
   STATUS[12].EXT.Operation := TRUE;
   STATUS[12].EXT.Forced := FALSE;
   STATUS[12].EXT.BIT29 := FALSE;
   STATUS[12].EXT.BIT30 := FALSE;
   STATUS[12].EXT.BIT31 := FALSE;
   STATUS[12].EXT.ModeBit1 := FALSE;
   STATUS[12].EXT.ModeBit2 := FALSE;
   STATUS[12].EXT.ModeBit3 := FALSE;
   STATUS[12].EXT.BIT19 := FALSE;
   STATUS[12].EXT.BIT20 := FALSE;
   STATUS[12].EXT.AlarmSuppressed := TRUE;
   STATUS[12].EXT.AlarmPrsent := FALSE;
   STATUS[12].EXT.AlarmFailUnAck := FALSE;
   STATUS[12].Status := 1;
   STATUS[12].TimeStamp := 16#3928;
   STATUS[13].VALUE := 0.0;
   STATUS[13].TRIGVALUE := 0.0;
   STATUS[13].EXT.AlarmWarnUnAck := TRUE;
   STATUS[13].EXT.AckRequired := FALSE;
   STATUS[13].EXT.Maintanence := FALSE;
   STATUS[13].EXT.Operation := TRUE;
   STATUS[13].EXT.Forced := FALSE;
   STATUS[13].EXT.BIT29 := FALSE;
   STATUS[13].EXT.BIT30 := FALSE;
   STATUS[13].EXT.BIT31 := FALSE;
   STATUS[13].EXT.ModeBit1 := FALSE;
   STATUS[13].EXT.ModeBit2 := FALSE;
   STATUS[13].EXT.ModeBit3 := FALSE;
   STATUS[13].EXT.BIT19 := FALSE;
   STATUS[13].EXT.BIT20 := FALSE;
   STATUS[13].EXT.AlarmSuppressed := TRUE;
   STATUS[13].EXT.AlarmPrsent := FALSE;
   STATUS[13].EXT.AlarmFailUnAck := FALSE;
   STATUS[13].Status := 1;
   STATUS[13].TimeStamp := 16#3928;
   STATUS[14].VALUE := 0.0;
   STATUS[14].TRIGVALUE := 3.9375;
   STATUS[14].EXT.AlarmWarnUnAck := TRUE;
   STATUS[14].EXT.AckRequired := FALSE;
   STATUS[14].EXT.Maintanence := FALSE;
   STATUS[14].EXT.Operation := TRUE;
   STATUS[14].EXT.Forced := FALSE;
   STATUS[14].EXT.BIT29 := FALSE;
   STATUS[14].EXT.BIT30 := FALSE;
   STATUS[14].EXT.BIT31 := FALSE;
   STATUS[14].EXT.ModeBit1 := FALSE;
   STATUS[14].EXT.ModeBit2 := FALSE;
   STATUS[14].EXT.ModeBit3 := FALSE;
   STATUS[14].EXT.BIT19 := FALSE;
   STATUS[14].EXT.BIT20 := FALSE;
   STATUS[14].EXT.AlarmSuppressed := FALSE;
   STATUS[14].EXT.AlarmPrsent := FALSE;
   STATUS[14].EXT.AlarmFailUnAck := FALSE;
   STATUS[14].Status := 1;
   STATUS[14].TimeStamp := 16#2756;
   STATUS[15].VALUE := 0.0;
   STATUS[15].TRIGVALUE := 3.9375;
   STATUS[15].EXT.AlarmWarnUnAck := TRUE;
   STATUS[15].EXT.AckRequired := FALSE;
   STATUS[15].EXT.Maintanence := FALSE;
   STATUS[15].EXT.Operation := TRUE;
   STATUS[15].EXT.Forced := FALSE;
   STATUS[15].EXT.BIT29 := FALSE;
   STATUS[15].EXT.BIT30 := FALSE;
   STATUS[15].EXT.BIT31 := FALSE;
   STATUS[15].EXT.ModeBit1 := FALSE;
   STATUS[15].EXT.ModeBit2 := FALSE;
   STATUS[15].EXT.ModeBit3 := FALSE;
   STATUS[15].EXT.BIT19 := FALSE;
   STATUS[15].EXT.BIT20 := FALSE;
   STATUS[15].EXT.AlarmSuppressed := FALSE;
   STATUS[15].EXT.AlarmPrsent := FALSE;
   STATUS[15].EXT.AlarmFailUnAck := FALSE;
   STATUS[15].Status := 1;
   STATUS[15].TimeStamp := 16#2756;
   STATUS[16].VALUE := 0.0;
   STATUS[16].TRIGVALUE := 0.0;
   STATUS[16].EXT.AlarmWarnUnAck := TRUE;
   STATUS[16].EXT.AckRequired := FALSE;
   STATUS[16].EXT.Maintanence := FALSE;
   STATUS[16].EXT.Operation := TRUE;
   STATUS[16].EXT.Forced := FALSE;
   STATUS[16].EXT.BIT29 := FALSE;
   STATUS[16].EXT.BIT30 := FALSE;
   STATUS[16].EXT.BIT31 := FALSE;
   STATUS[16].EXT.ModeBit1 := FALSE;
   STATUS[16].EXT.ModeBit2 := FALSE;
   STATUS[16].EXT.ModeBit3 := FALSE;
   STATUS[16].EXT.BIT19 := FALSE;
   STATUS[16].EXT.BIT20 := FALSE;
   STATUS[16].EXT.AlarmSuppressed := FALSE;
   STATUS[16].EXT.AlarmPrsent := FALSE;
   STATUS[16].EXT.AlarmFailUnAck := FALSE;
   STATUS[16].Status := 1;
   STATUS[16].TimeStamp := 16#3928;
   STATUS[17].VALUE := 9.175245E-37;
   STATUS[17].TRIGVALUE := 100.7218;
   STATUS[17].EXT.AlarmWarnUnAck := TRUE;
   STATUS[17].EXT.AckRequired := FALSE;
   STATUS[17].EXT.Maintanence := FALSE;
   STATUS[17].EXT.Operation := TRUE;
   STATUS[17].EXT.Forced := FALSE;
   STATUS[17].EXT.BIT29 := FALSE;
   STATUS[17].EXT.BIT30 := FALSE;
   STATUS[17].EXT.BIT31 := FALSE;
   STATUS[17].EXT.ModeBit1 := FALSE;
   STATUS[17].EXT.ModeBit2 := FALSE;
   STATUS[17].EXT.ModeBit3 := FALSE;
   STATUS[17].EXT.BIT19 := FALSE;
   STATUS[17].EXT.BIT20 := FALSE;
   STATUS[17].EXT.AlarmSuppressed := FALSE;
   STATUS[17].EXT.AlarmPrsent := FALSE;
   STATUS[17].EXT.AlarmFailUnAck := FALSE;
   STATUS[17].Status := 1;
   STATUS[17].TimeStamp := 16#32A0;
   STATUS[18].VALUE := -118.5185;
   STATUS[18].TRIGVALUE := -118.5185;
   STATUS[18].EXT.AlarmWarnUnAck := TRUE;
   STATUS[18].EXT.AckRequired := FALSE;
   STATUS[18].EXT.Maintanence := FALSE;
   STATUS[18].EXT.Operation := TRUE;
   STATUS[18].EXT.Forced := FALSE;
   STATUS[18].EXT.BIT29 := FALSE;
   STATUS[18].EXT.BIT30 := FALSE;
   STATUS[18].EXT.BIT31 := FALSE;
   STATUS[18].EXT.ModeBit1 := FALSE;
   STATUS[18].EXT.ModeBit2 := FALSE;
   STATUS[18].EXT.ModeBit3 := FALSE;
   STATUS[18].EXT.BIT19 := FALSE;
   STATUS[18].EXT.BIT20 := FALSE;
   STATUS[18].EXT.AlarmSuppressed := FALSE;
   STATUS[18].EXT.AlarmPrsent := FALSE;
   STATUS[18].EXT.AlarmFailUnAck := FALSE;
   STATUS[18].Status := 1;
   STATUS[18].TimeStamp := 16#D02B;
   STATUS[19].VALUE := 38.75868;
   STATUS[19].TRIGVALUE := -85.46368;
   STATUS[19].EXT.AlarmWarnUnAck := TRUE;
   STATUS[19].EXT.AckRequired := FALSE;
   STATUS[19].EXT.Maintanence := FALSE;
   STATUS[19].EXT.Operation := TRUE;
   STATUS[19].EXT.Forced := FALSE;
   STATUS[19].EXT.BIT29 := FALSE;
   STATUS[19].EXT.BIT30 := FALSE;
   STATUS[19].EXT.BIT31 := FALSE;
   STATUS[19].EXT.ModeBit1 := FALSE;
   STATUS[19].EXT.ModeBit2 := FALSE;
   STATUS[19].EXT.ModeBit3 := FALSE;
   STATUS[19].EXT.BIT19 := FALSE;
   STATUS[19].EXT.BIT20 := FALSE;
   STATUS[19].EXT.AlarmSuppressed := TRUE;
   STATUS[19].EXT.AlarmPrsent := FALSE;
   STATUS[19].EXT.AlarmFailUnAck := FALSE;
   STATUS[19].Status := 1;
   STATUS[19].TimeStamp := 16#CFE1;
   STATUS[20].VALUE := 38.8491;
   STATUS[20].TRIGVALUE := -72.46094;
   STATUS[20].EXT.AlarmWarnUnAck := TRUE;
   STATUS[20].EXT.AckRequired := FALSE;
   STATUS[20].EXT.Maintanence := FALSE;
   STATUS[20].EXT.Operation := TRUE;
   STATUS[20].EXT.Forced := FALSE;
   STATUS[20].EXT.BIT29 := FALSE;
   STATUS[20].EXT.BIT30 := FALSE;
   STATUS[20].EXT.BIT31 := FALSE;
   STATUS[20].EXT.ModeBit1 := FALSE;
   STATUS[20].EXT.ModeBit2 := FALSE;
   STATUS[20].EXT.ModeBit3 := FALSE;
   STATUS[20].EXT.BIT19 := FALSE;
   STATUS[20].EXT.BIT20 := FALSE;
   STATUS[20].EXT.AlarmSuppressed := TRUE;
   STATUS[20].EXT.AlarmPrsent := FALSE;
   STATUS[20].EXT.AlarmFailUnAck := FALSE;
   STATUS[20].Status := 1;
   STATUS[20].TimeStamp := 16#CFE8;
   STATUS[21].VALUE := 46.21853;
   STATUS[21].TRIGVALUE := -68.2382;
   STATUS[21].EXT.AlarmWarnUnAck := TRUE;
   STATUS[21].EXT.AckRequired := FALSE;
   STATUS[21].EXT.Maintanence := FALSE;
   STATUS[21].EXT.Operation := TRUE;
   STATUS[21].EXT.Forced := FALSE;
   STATUS[21].EXT.BIT29 := FALSE;
   STATUS[21].EXT.BIT30 := FALSE;
   STATUS[21].EXT.BIT31 := FALSE;
   STATUS[21].EXT.ModeBit1 := FALSE;
   STATUS[21].EXT.ModeBit2 := FALSE;
   STATUS[21].EXT.ModeBit3 := FALSE;
   STATUS[21].EXT.BIT19 := FALSE;
   STATUS[21].EXT.BIT20 := FALSE;
   STATUS[21].EXT.AlarmSuppressed := TRUE;
   STATUS[21].EXT.AlarmPrsent := FALSE;
   STATUS[21].EXT.AlarmFailUnAck := FALSE;
   STATUS[21].Status := 1;
   STATUS[21].TimeStamp := 16#CFEE;
   STATUS[22].VALUE := 46.82436;
   STATUS[22].TRIGVALUE := -65.98669;
   STATUS[22].EXT.AlarmWarnUnAck := TRUE;
   STATUS[22].EXT.AckRequired := FALSE;
   STATUS[22].EXT.Maintanence := FALSE;
   STATUS[22].EXT.Operation := TRUE;
   STATUS[22].EXT.Forced := FALSE;
   STATUS[22].EXT.BIT29 := FALSE;
   STATUS[22].EXT.BIT30 := FALSE;
   STATUS[22].EXT.BIT31 := FALSE;
   STATUS[22].EXT.ModeBit1 := FALSE;
   STATUS[22].EXT.ModeBit2 := FALSE;
   STATUS[22].EXT.ModeBit3 := FALSE;
   STATUS[22].EXT.BIT19 := FALSE;
   STATUS[22].EXT.BIT20 := FALSE;
   STATUS[22].EXT.AlarmSuppressed := TRUE;
   STATUS[22].EXT.AlarmPrsent := FALSE;
   STATUS[22].EXT.AlarmFailUnAck := FALSE;
   STATUS[22].Status := 1;
   STATUS[22].TimeStamp := 16#CFF3;
   STATUS[23].VALUE := 94.6506;
   STATUS[23].TRIGVALUE := 94.01041;
   STATUS[23].EXT.AlarmWarnUnAck := TRUE;
   STATUS[23].EXT.AckRequired := FALSE;
   STATUS[23].EXT.Maintanence := FALSE;
   STATUS[23].EXT.Operation := TRUE;
   STATUS[23].EXT.Forced := FALSE;
   STATUS[23].EXT.BIT29 := FALSE;
   STATUS[23].EXT.BIT30 := FALSE;
   STATUS[23].EXT.BIT31 := FALSE;
   STATUS[23].EXT.ModeBit1 := FALSE;
   STATUS[23].EXT.ModeBit2 := FALSE;
   STATUS[23].EXT.ModeBit3 := FALSE;
   STATUS[23].EXT.BIT19 := FALSE;
   STATUS[23].EXT.BIT20 := FALSE;
   STATUS[23].EXT.AlarmSuppressed := FALSE;
   STATUS[23].EXT.AlarmPrsent := FALSE;
   STATUS[23].EXT.AlarmFailUnAck := FALSE;
   STATUS[23].Status := 1;
   STATUS[23].TimeStamp := 16#BAFA;
   STATUS[24].VALUE := 6.610245;
   STATUS[24].TRIGVALUE := 0.0;
   STATUS[24].EXT.AlarmWarnUnAck := TRUE;
   STATUS[24].EXT.AckRequired := FALSE;
   STATUS[24].EXT.Maintanence := FALSE;
   STATUS[24].EXT.Operation := TRUE;
   STATUS[24].EXT.Forced := FALSE;
   STATUS[24].EXT.BIT29 := FALSE;
   STATUS[24].EXT.BIT30 := FALSE;
   STATUS[24].EXT.BIT31 := FALSE;
   STATUS[24].EXT.ModeBit1 := FALSE;
   STATUS[24].EXT.ModeBit2 := FALSE;
   STATUS[24].EXT.ModeBit3 := FALSE;
   STATUS[24].EXT.BIT19 := FALSE;
   STATUS[24].EXT.BIT20 := FALSE;
   STATUS[24].EXT.AlarmSuppressed := TRUE;
   STATUS[24].EXT.AlarmPrsent := FALSE;
   STATUS[24].EXT.AlarmFailUnAck := FALSE;
   STATUS[24].Status := 1;
   STATUS[24].TimeStamp := 16#3928;
   STATUS[25].VALUE := 0.0;
   STATUS[25].TRIGVALUE := 0.0;
   STATUS[25].EXT.AlarmWarnUnAck := TRUE;
   STATUS[25].EXT.AckRequired := FALSE;
   STATUS[25].EXT.Maintanence := FALSE;
   STATUS[25].EXT.Operation := TRUE;
   STATUS[25].EXT.Forced := TRUE;
   STATUS[25].EXT.BIT29 := FALSE;
   STATUS[25].EXT.BIT30 := FALSE;
   STATUS[25].EXT.BIT31 := FALSE;
   STATUS[25].EXT.ModeBit1 := FALSE;
   STATUS[25].EXT.ModeBit2 := FALSE;
   STATUS[25].EXT.ModeBit3 := FALSE;
   STATUS[25].EXT.BIT19 := FALSE;
   STATUS[25].EXT.BIT20 := FALSE;
   STATUS[25].EXT.AlarmSuppressed := TRUE;
   STATUS[25].EXT.AlarmPrsent := FALSE;
   STATUS[25].EXT.AlarmFailUnAck := FALSE;
   STATUS[25].Status := 1;
   STATUS[25].TimeStamp := 16#3928;
   STATUS[26].VALUE := 8.242188;
   STATUS[26].TRIGVALUE := 5.99826;
   STATUS[26].EXT.AlarmWarnUnAck := TRUE;
   STATUS[26].EXT.AckRequired := FALSE;
   STATUS[26].EXT.Maintanence := FALSE;
   STATUS[26].EXT.Operation := TRUE;
   STATUS[26].EXT.Forced := FALSE;
   STATUS[26].EXT.BIT29 := FALSE;
   STATUS[26].EXT.BIT30 := FALSE;
   STATUS[26].EXT.BIT31 := FALSE;
   STATUS[26].EXT.ModeBit1 := FALSE;
   STATUS[26].EXT.ModeBit2 := FALSE;
   STATUS[26].EXT.ModeBit3 := FALSE;
   STATUS[26].EXT.BIT19 := FALSE;
   STATUS[26].EXT.BIT20 := FALSE;
   STATUS[26].EXT.AlarmSuppressed := FALSE;
   STATUS[26].EXT.AlarmPrsent := FALSE;
   STATUS[26].EXT.AlarmFailUnAck := FALSE;
   STATUS[26].Status := 1;
   STATUS[26].TimeStamp := 16#E969;
   STATUS[27].VALUE := 97.4754;
   STATUS[27].TRIGVALUE := 73.09389;
   STATUS[27].EXT.AlarmWarnUnAck := TRUE;
   STATUS[27].EXT.AckRequired := FALSE;
   STATUS[27].EXT.Maintanence := FALSE;
   STATUS[27].EXT.Operation := TRUE;
   STATUS[27].EXT.Forced := FALSE;
   STATUS[27].EXT.BIT29 := FALSE;
   STATUS[27].EXT.BIT30 := FALSE;
   STATUS[27].EXT.BIT31 := FALSE;
   STATUS[27].EXT.ModeBit1 := FALSE;
   STATUS[27].EXT.ModeBit2 := FALSE;
   STATUS[27].EXT.ModeBit3 := FALSE;
   STATUS[27].EXT.BIT19 := FALSE;
   STATUS[27].EXT.BIT20 := FALSE;
   STATUS[27].EXT.AlarmSuppressed := TRUE;
   STATUS[27].EXT.AlarmPrsent := FALSE;
   STATUS[27].EXT.AlarmFailUnAck := FALSE;
   STATUS[27].Status := 1;
   STATUS[27].TimeStamp := 16#0B2D;
   STATUS[28].VALUE := 87.21065;
   STATUS[28].TRIGVALUE := 72.46455;
   STATUS[28].EXT.AlarmWarnUnAck := TRUE;
   STATUS[28].EXT.AckRequired := FALSE;
   STATUS[28].EXT.Maintanence := FALSE;
   STATUS[28].EXT.Operation := TRUE;
   STATUS[28].EXT.Forced := FALSE;
   STATUS[28].EXT.BIT29 := FALSE;
   STATUS[28].EXT.BIT30 := FALSE;
   STATUS[28].EXT.BIT31 := FALSE;
   STATUS[28].EXT.ModeBit1 := FALSE;
   STATUS[28].EXT.ModeBit2 := FALSE;
   STATUS[28].EXT.ModeBit3 := FALSE;
   STATUS[28].EXT.BIT19 := FALSE;
   STATUS[28].EXT.BIT20 := FALSE;
   STATUS[28].EXT.AlarmSuppressed := TRUE;
   STATUS[28].EXT.AlarmPrsent := FALSE;
   STATUS[28].EXT.AlarmFailUnAck := FALSE;
   STATUS[28].Status := 1;
   STATUS[28].TimeStamp := 16#2CB5;
   STATUS[29].VALUE := 0.0;
   STATUS[29].TRIGVALUE := 0.0;
   STATUS[29].EXT.AlarmWarnUnAck := TRUE;
   STATUS[29].EXT.AckRequired := FALSE;
   STATUS[29].EXT.Maintanence := FALSE;
   STATUS[29].EXT.Operation := TRUE;
   STATUS[29].EXT.Forced := FALSE;
   STATUS[29].EXT.BIT29 := FALSE;
   STATUS[29].EXT.BIT30 := FALSE;
   STATUS[29].EXT.BIT31 := FALSE;
   STATUS[29].EXT.ModeBit1 := FALSE;
   STATUS[29].EXT.ModeBit2 := FALSE;
   STATUS[29].EXT.ModeBit3 := FALSE;
   STATUS[29].EXT.BIT19 := FALSE;
   STATUS[29].EXT.BIT20 := FALSE;
   STATUS[29].EXT.AlarmSuppressed := TRUE;
   STATUS[29].EXT.AlarmPrsent := FALSE;
   STATUS[29].EXT.AlarmFailUnAck := FALSE;
   STATUS[29].Status := 1;
   STATUS[29].TimeStamp := 16#3928;
   STATUS[30].VALUE := 0.0;
   STATUS[30].TRIGVALUE := 0.0;
   STATUS[30].EXT.AlarmWarnUnAck := TRUE;
   STATUS[30].EXT.AckRequired := FALSE;
   STATUS[30].EXT.Maintanence := FALSE;
   STATUS[30].EXT.Operation := TRUE;
   STATUS[30].EXT.Forced := FALSE;
   STATUS[30].EXT.BIT29 := FALSE;
   STATUS[30].EXT.BIT30 := FALSE;
   STATUS[30].EXT.BIT31 := FALSE;
   STATUS[30].EXT.ModeBit1 := FALSE;
   STATUS[30].EXT.ModeBit2 := FALSE;
   STATUS[30].EXT.ModeBit3 := FALSE;
   STATUS[30].EXT.BIT19 := FALSE;
   STATUS[30].EXT.BIT20 := FALSE;
   STATUS[30].EXT.AlarmSuppressed := TRUE;
   STATUS[30].EXT.AlarmPrsent := FALSE;
   STATUS[30].EXT.AlarmFailUnAck := FALSE;
   STATUS[30].Status := 1;
   STATUS[30].TimeStamp := 16#3928;
   STATUS[31].VALUE := 0.0;
   STATUS[31].TRIGVALUE := 0.0;
   STATUS[31].EXT.AlarmWarnUnAck := TRUE;
   STATUS[31].EXT.AckRequired := FALSE;
   STATUS[31].EXT.Maintanence := FALSE;
   STATUS[31].EXT.Operation := TRUE;
   STATUS[31].EXT.Forced := FALSE;
   STATUS[31].EXT.BIT29 := FALSE;
   STATUS[31].EXT.BIT30 := FALSE;
   STATUS[31].EXT.BIT31 := FALSE;
   STATUS[31].EXT.ModeBit1 := FALSE;
   STATUS[31].EXT.ModeBit2 := FALSE;
   STATUS[31].EXT.ModeBit3 := FALSE;
   STATUS[31].EXT.BIT19 := FALSE;
   STATUS[31].EXT.BIT20 := FALSE;
   STATUS[31].EXT.AlarmSuppressed := TRUE;
   STATUS[31].EXT.AlarmPrsent := FALSE;
   STATUS[31].EXT.AlarmFailUnAck := FALSE;
   STATUS[31].Status := 1;
   STATUS[31].TimeStamp := 16#3928;
   STATUS[32].VALUE := 0.0;
   STATUS[32].TRIGVALUE := 0.0;
   STATUS[32].EXT.AlarmWarnUnAck := TRUE;
   STATUS[32].EXT.AckRequired := FALSE;
   STATUS[32].EXT.Maintanence := FALSE;
   STATUS[32].EXT.Operation := TRUE;
   STATUS[32].EXT.Forced := FALSE;
   STATUS[32].EXT.BIT29 := FALSE;
   STATUS[32].EXT.BIT30 := FALSE;
   STATUS[32].EXT.BIT31 := FALSE;
   STATUS[32].EXT.ModeBit1 := FALSE;
   STATUS[32].EXT.ModeBit2 := FALSE;
   STATUS[32].EXT.ModeBit3 := FALSE;
   STATUS[32].EXT.BIT19 := FALSE;
   STATUS[32].EXT.BIT20 := FALSE;
   STATUS[32].EXT.AlarmSuppressed := TRUE;
   STATUS[32].EXT.AlarmPrsent := FALSE;
   STATUS[32].EXT.AlarmFailUnAck := FALSE;
   STATUS[32].Status := 1;
   STATUS[32].TimeStamp := 16#3928;
   STATUS[33].VALUE := 0.0;
   STATUS[33].TRIGVALUE := 0.0;
   STATUS[33].EXT.AlarmWarnUnAck := TRUE;
   STATUS[33].EXT.AckRequired := FALSE;
   STATUS[33].EXT.Maintanence := FALSE;
   STATUS[33].EXT.Operation := TRUE;
   STATUS[33].EXT.Forced := FALSE;
   STATUS[33].EXT.BIT29 := FALSE;
   STATUS[33].EXT.BIT30 := FALSE;
   STATUS[33].EXT.BIT31 := FALSE;
   STATUS[33].EXT.ModeBit1 := FALSE;
   STATUS[33].EXT.ModeBit2 := FALSE;
   STATUS[33].EXT.ModeBit3 := FALSE;
   STATUS[33].EXT.BIT19 := FALSE;
   STATUS[33].EXT.BIT20 := FALSE;
   STATUS[33].EXT.AlarmSuppressed := TRUE;
   STATUS[33].EXT.AlarmPrsent := FALSE;
   STATUS[33].EXT.AlarmFailUnAck := FALSE;
   STATUS[33].Status := 1;
   STATUS[33].TimeStamp := 16#3928;
   STATUS[34].VALUE := 0.0;
   STATUS[34].TRIGVALUE := 0.0;
   STATUS[34].EXT.AlarmWarnUnAck := TRUE;
   STATUS[34].EXT.AckRequired := FALSE;
   STATUS[34].EXT.Maintanence := FALSE;
   STATUS[34].EXT.Operation := TRUE;
   STATUS[34].EXT.Forced := FALSE;
   STATUS[34].EXT.BIT29 := FALSE;
   STATUS[34].EXT.BIT30 := FALSE;
   STATUS[34].EXT.BIT31 := FALSE;
   STATUS[34].EXT.ModeBit1 := FALSE;
   STATUS[34].EXT.ModeBit2 := FALSE;
   STATUS[34].EXT.ModeBit3 := FALSE;
   STATUS[34].EXT.BIT19 := FALSE;
   STATUS[34].EXT.BIT20 := FALSE;
   STATUS[34].EXT.AlarmSuppressed := TRUE;
   STATUS[34].EXT.AlarmPrsent := FALSE;
   STATUS[34].EXT.AlarmFailUnAck := FALSE;
   STATUS[34].Status := 1;
   STATUS[34].TimeStamp := 16#3928;
   STATUS[35].VALUE := -0.03255209;
   STATUS[35].TRIGVALUE := 144.2634;
   STATUS[35].EXT.AlarmWarnUnAck := TRUE;
   STATUS[35].EXT.AckRequired := FALSE;
   STATUS[35].EXT.Maintanence := FALSE;
   STATUS[35].EXT.Operation := TRUE;
   STATUS[35].EXT.Forced := FALSE;
   STATUS[35].EXT.BIT29 := FALSE;
   STATUS[35].EXT.BIT30 := FALSE;
   STATUS[35].EXT.BIT31 := FALSE;
   STATUS[35].EXT.ModeBit1 := FALSE;
   STATUS[35].EXT.ModeBit2 := FALSE;
   STATUS[35].EXT.ModeBit3 := FALSE;
   STATUS[35].EXT.BIT19 := FALSE;
   STATUS[35].EXT.BIT20 := FALSE;
   STATUS[35].EXT.AlarmSuppressed := TRUE;
   STATUS[35].EXT.AlarmPrsent := FALSE;
   STATUS[35].EXT.AlarmFailUnAck := FALSE;
   STATUS[35].Status := 1;
   STATUS[35].TimeStamp := 16#DF93;
   STATUS[36].VALUE := 24.66105;
   STATUS[36].TRIGVALUE := 80.89346;
   STATUS[36].EXT.AlarmWarnUnAck := TRUE;
   STATUS[36].EXT.AckRequired := FALSE;
   STATUS[36].EXT.Maintanence := FALSE;
   STATUS[36].EXT.Operation := TRUE;
   STATUS[36].EXT.Forced := FALSE;
   STATUS[36].EXT.BIT29 := FALSE;
   STATUS[36].EXT.BIT30 := FALSE;
   STATUS[36].EXT.BIT31 := FALSE;
   STATUS[36].EXT.ModeBit1 := FALSE;
   STATUS[36].EXT.ModeBit2 := FALSE;
   STATUS[36].EXT.ModeBit3 := FALSE;
   STATUS[36].EXT.BIT19 := FALSE;
   STATUS[36].EXT.BIT20 := FALSE;
   STATUS[36].EXT.AlarmSuppressed := TRUE;
   STATUS[36].EXT.AlarmPrsent := FALSE;
   STATUS[36].EXT.AlarmFailUnAck := FALSE;
   STATUS[36].Status := 1;
   STATUS[36].TimeStamp := 16#6A1D;
   STATUS[37].VALUE := -177.7778;
   STATUS[37].TRIGVALUE := -177.7778;
   STATUS[37].EXT.AlarmWarnUnAck := FALSE;
   STATUS[37].EXT.AckRequired := FALSE;
   STATUS[37].EXT.Maintanence := FALSE;
   STATUS[37].EXT.Operation := TRUE;
   STATUS[37].EXT.Forced := FALSE;
   STATUS[37].EXT.BIT29 := FALSE;
   STATUS[37].EXT.BIT30 := FALSE;
   STATUS[37].EXT.BIT31 := FALSE;
   STATUS[37].EXT.ModeBit1 := FALSE;
   STATUS[37].EXT.ModeBit2 := FALSE;
   STATUS[37].EXT.ModeBit3 := FALSE;
   STATUS[37].EXT.BIT19 := FALSE;
   STATUS[37].EXT.BIT20 := FALSE;
   STATUS[37].EXT.AlarmSuppressed := TRUE;
   STATUS[37].EXT.AlarmPrsent := TRUE;
   STATUS[37].EXT.AlarmFailUnAck := TRUE;
   STATUS[37].Status := 150;
   STATUS[37].TimeStamp := 16#9344;
   STATUS[38].VALUE := -0.2589699;
   STATUS[38].TRIGVALUE := -0.2633102;
   STATUS[38].EXT.AlarmWarnUnAck := FALSE;
   STATUS[38].EXT.AckRequired := FALSE;
   STATUS[38].EXT.Maintanence := FALSE;
   STATUS[38].EXT.Operation := TRUE;
   STATUS[38].EXT.Forced := FALSE;
   STATUS[38].EXT.BIT29 := FALSE;
   STATUS[38].EXT.BIT30 := FALSE;
   STATUS[38].EXT.BIT31 := FALSE;
   STATUS[38].EXT.ModeBit1 := FALSE;
   STATUS[38].EXT.ModeBit2 := FALSE;
   STATUS[38].EXT.ModeBit3 := FALSE;
   STATUS[38].EXT.BIT19 := FALSE;
   STATUS[38].EXT.BIT20 := FALSE;
   STATUS[38].EXT.AlarmSuppressed := TRUE;
   STATUS[38].EXT.AlarmPrsent := TRUE;
   STATUS[38].EXT.AlarmFailUnAck := TRUE;
   STATUS[38].Status := 176;
   STATUS[38].TimeStamp := 16#84E5;
   STATUS[39].VALUE := 6.475695;
   STATUS[39].TRIGVALUE := -0.01041667;
   STATUS[39].EXT.AlarmWarnUnAck := TRUE;
   STATUS[39].EXT.AckRequired := FALSE;
   STATUS[39].EXT.Maintanence := FALSE;
   STATUS[39].EXT.Operation := TRUE;
   STATUS[39].EXT.Forced := FALSE;
   STATUS[39].EXT.BIT29 := FALSE;
   STATUS[39].EXT.BIT30 := FALSE;
   STATUS[39].EXT.BIT31 := FALSE;
   STATUS[39].EXT.ModeBit1 := FALSE;
   STATUS[39].EXT.ModeBit2 := FALSE;
   STATUS[39].EXT.ModeBit3 := FALSE;
   STATUS[39].EXT.BIT19 := FALSE;
   STATUS[39].EXT.BIT20 := FALSE;
   STATUS[39].EXT.AlarmSuppressed := TRUE;
   STATUS[39].EXT.AlarmPrsent := FALSE;
   STATUS[39].EXT.AlarmFailUnAck := FALSE;
   STATUS[39].Status := 1;
   STATUS[39].TimeStamp := 16#3838;
   STATUS[40].VALUE := 5.940393;
   STATUS[40].TRIGVALUE := 5.9375;
   STATUS[40].EXT.AlarmWarnUnAck := FALSE;
   STATUS[40].EXT.AckRequired := FALSE;
   STATUS[40].EXT.Maintanence := FALSE;
   STATUS[40].EXT.Operation := TRUE;
   STATUS[40].EXT.Forced := FALSE;
   STATUS[40].EXT.BIT29 := FALSE;
   STATUS[40].EXT.BIT30 := FALSE;
   STATUS[40].EXT.BIT31 := FALSE;
   STATUS[40].EXT.ModeBit1 := FALSE;
   STATUS[40].EXT.ModeBit2 := FALSE;
   STATUS[40].EXT.ModeBit3 := FALSE;
   STATUS[40].EXT.BIT19 := FALSE;
   STATUS[40].EXT.BIT20 := FALSE;
   STATUS[40].EXT.AlarmSuppressed := TRUE;
   STATUS[40].EXT.AlarmPrsent := TRUE;
   STATUS[40].EXT.AlarmFailUnAck := TRUE;
   STATUS[40].Status := 176;
   STATUS[40].TimeStamp := 16#84E5;
   STATUS[41].VALUE := 71.0;
   STATUS[41].TRIGVALUE := 0.5177951;
   STATUS[41].EXT.AlarmWarnUnAck := TRUE;
   STATUS[41].EXT.AckRequired := FALSE;
   STATUS[41].EXT.Maintanence := FALSE;
   STATUS[41].EXT.Operation := TRUE;
   STATUS[41].EXT.Forced := FALSE;
   STATUS[41].EXT.BIT29 := FALSE;
   STATUS[41].EXT.BIT30 := FALSE;
   STATUS[41].EXT.BIT31 := FALSE;
   STATUS[41].EXT.ModeBit1 := FALSE;
   STATUS[41].EXT.ModeBit2 := FALSE;
   STATUS[41].EXT.ModeBit3 := FALSE;
   STATUS[41].EXT.BIT19 := FALSE;
   STATUS[41].EXT.BIT20 := FALSE;
   STATUS[41].EXT.AlarmSuppressed := TRUE;
   STATUS[41].EXT.AlarmPrsent := FALSE;
   STATUS[41].EXT.AlarmFailUnAck := FALSE;
   STATUS[41].Status := 1;
   STATUS[41].TimeStamp := 16#B051;
   STATUS[42].VALUE := 1.88151;
   STATUS[42].TRIGVALUE := 1.768663;
   STATUS[42].EXT.AlarmWarnUnAck := FALSE;
   STATUS[42].EXT.AckRequired := FALSE;
   STATUS[42].EXT.Maintanence := FALSE;
   STATUS[42].EXT.Operation := TRUE;
   STATUS[42].EXT.Forced := FALSE;
   STATUS[42].EXT.BIT29 := FALSE;
   STATUS[42].EXT.BIT30 := FALSE;
   STATUS[42].EXT.BIT31 := FALSE;
   STATUS[42].EXT.ModeBit1 := FALSE;
   STATUS[42].EXT.ModeBit2 := FALSE;
   STATUS[42].EXT.ModeBit3 := FALSE;
   STATUS[42].EXT.BIT19 := FALSE;
   STATUS[42].EXT.BIT20 := FALSE;
   STATUS[42].EXT.AlarmSuppressed := TRUE;
   STATUS[42].EXT.AlarmPrsent := TRUE;
   STATUS[42].EXT.AlarmFailUnAck := TRUE;
   STATUS[42].Status := 176;
   STATUS[42].TimeStamp := 16#84E5;
   STATUS[43].VALUE := 5.918693;
   STATUS[43].TRIGVALUE := 4.895834;
   STATUS[43].EXT.AlarmWarnUnAck := TRUE;
   STATUS[43].EXT.AckRequired := FALSE;
   STATUS[43].EXT.Maintanence := FALSE;
   STATUS[43].EXT.Operation := TRUE;
   STATUS[43].EXT.Forced := FALSE;
   STATUS[43].EXT.BIT29 := FALSE;
   STATUS[43].EXT.BIT30 := FALSE;
   STATUS[43].EXT.BIT31 := FALSE;
   STATUS[43].EXT.ModeBit1 := FALSE;
   STATUS[43].EXT.ModeBit2 := FALSE;
   STATUS[43].EXT.ModeBit3 := FALSE;
   STATUS[43].EXT.BIT19 := FALSE;
   STATUS[43].EXT.BIT20 := FALSE;
   STATUS[43].EXT.AlarmSuppressed := TRUE;
   STATUS[43].EXT.AlarmPrsent := FALSE;
   STATUS[43].EXT.AlarmFailUnAck := FALSE;
   STATUS[43].Status := 1;
   STATUS[43].TimeStamp := 16#BD5F;
   STATUS[44].VALUE := -53.33333;
   STATUS[44].TRIGVALUE := -53.33333;
   STATUS[44].EXT.AlarmWarnUnAck := FALSE;
   STATUS[44].EXT.AckRequired := FALSE;
   STATUS[44].EXT.Maintanence := FALSE;
   STATUS[44].EXT.Operation := TRUE;
   STATUS[44].EXT.Forced := FALSE;
   STATUS[44].EXT.BIT29 := FALSE;
   STATUS[44].EXT.BIT30 := FALSE;
   STATUS[44].EXT.BIT31 := FALSE;
   STATUS[44].EXT.ModeBit1 := FALSE;
   STATUS[44].EXT.ModeBit2 := FALSE;
   STATUS[44].EXT.ModeBit3 := FALSE;
   STATUS[44].EXT.BIT19 := FALSE;
   STATUS[44].EXT.BIT20 := FALSE;
   STATUS[44].EXT.AlarmSuppressed := TRUE;
   STATUS[44].EXT.AlarmPrsent := TRUE;
   STATUS[44].EXT.AlarmFailUnAck := TRUE;
   STATUS[44].Status := 150;
   STATUS[44].TimeStamp := 16#9344;
   STATUS[45].VALUE := 118.7373;
   STATUS[45].TRIGVALUE := 0.0;
   STATUS[45].EXT.AlarmWarnUnAck := TRUE;
   STATUS[45].EXT.AckRequired := FALSE;
   STATUS[45].EXT.Maintanence := FALSE;
   STATUS[45].EXT.Operation := TRUE;
   STATUS[45].EXT.Forced := FALSE;
   STATUS[45].EXT.BIT29 := FALSE;
   STATUS[45].EXT.BIT30 := FALSE;
   STATUS[45].EXT.BIT31 := FALSE;
   STATUS[45].EXT.ModeBit1 := FALSE;
   STATUS[45].EXT.ModeBit2 := FALSE;
   STATUS[45].EXT.ModeBit3 := FALSE;
   STATUS[45].EXT.BIT19 := FALSE;
   STATUS[45].EXT.BIT20 := FALSE;
   STATUS[45].EXT.AlarmSuppressed := TRUE;
   STATUS[45].EXT.AlarmPrsent := FALSE;
   STATUS[45].EXT.AlarmFailUnAck := FALSE;
   STATUS[45].Status := 1;
   STATUS[45].TimeStamp := 16#3928;
   STATUS[46].VALUE := 39.898;
   STATUS[46].TRIGVALUE := 0.7790799;
   STATUS[46].EXT.AlarmWarnUnAck := TRUE;
   STATUS[46].EXT.AckRequired := FALSE;
   STATUS[46].EXT.Maintanence := FALSE;
   STATUS[46].EXT.Operation := TRUE;
   STATUS[46].EXT.Forced := FALSE;
   STATUS[46].EXT.BIT29 := FALSE;
   STATUS[46].EXT.BIT30 := FALSE;
   STATUS[46].EXT.BIT31 := FALSE;
   STATUS[46].EXT.ModeBit1 := FALSE;
   STATUS[46].EXT.ModeBit2 := FALSE;
   STATUS[46].EXT.ModeBit3 := FALSE;
   STATUS[46].EXT.BIT19 := FALSE;
   STATUS[46].EXT.BIT20 := FALSE;
   STATUS[46].EXT.AlarmSuppressed := TRUE;
   STATUS[46].EXT.AlarmPrsent := FALSE;
   STATUS[46].EXT.AlarmFailUnAck := FALSE;
   STATUS[46].Status := 1;
   STATUS[46].TimeStamp := 16#7392;
   STATUS[47].VALUE := 0.0;
   STATUS[47].TRIGVALUE := 0.0;
   STATUS[47].EXT.AlarmWarnUnAck := TRUE;
   STATUS[47].EXT.AckRequired := FALSE;
   STATUS[47].EXT.Maintanence := FALSE;
   STATUS[47].EXT.Operation := TRUE;
   STATUS[47].EXT.Forced := FALSE;
   STATUS[47].EXT.BIT29 := FALSE;
   STATUS[47].EXT.BIT30 := FALSE;
   STATUS[47].EXT.BIT31 := FALSE;
   STATUS[47].EXT.ModeBit1 := FALSE;
   STATUS[47].EXT.ModeBit2 := FALSE;
   STATUS[47].EXT.ModeBit3 := FALSE;
   STATUS[47].EXT.BIT19 := FALSE;
   STATUS[47].EXT.BIT20 := FALSE;
   STATUS[47].EXT.AlarmSuppressed := TRUE;
   STATUS[47].EXT.AlarmPrsent := FALSE;
   STATUS[47].EXT.AlarmFailUnAck := FALSE;
   STATUS[47].Status := 1;
   STATUS[47].TimeStamp := 16#3928;
   STATUS[48].VALUE := -11.85185;
   STATUS[48].TRIGVALUE := -11.85185;
   STATUS[48].EXT.AlarmWarnUnAck := FALSE;
   STATUS[48].EXT.AckRequired := FALSE;
   STATUS[48].EXT.Maintanence := FALSE;
   STATUS[48].EXT.Operation := TRUE;
   STATUS[48].EXT.Forced := FALSE;
   STATUS[48].EXT.BIT29 := FALSE;
   STATUS[48].EXT.BIT30 := FALSE;
   STATUS[48].EXT.BIT31 := FALSE;
   STATUS[48].EXT.ModeBit1 := FALSE;
   STATUS[48].EXT.ModeBit2 := FALSE;
   STATUS[48].EXT.ModeBit3 := FALSE;
   STATUS[48].EXT.BIT19 := FALSE;
   STATUS[48].EXT.BIT20 := FALSE;
   STATUS[48].EXT.AlarmSuppressed := TRUE;
   STATUS[48].EXT.AlarmPrsent := TRUE;
   STATUS[48].EXT.AlarmFailUnAck := TRUE;
   STATUS[48].Status := 150;
   STATUS[48].TimeStamp := 16#9344;
   STATUS[49].VALUE := 0.0;
   STATUS[49].TRIGVALUE := 0.0;
   STATUS[49].EXT.AlarmWarnUnAck := TRUE;
   STATUS[49].EXT.AckRequired := FALSE;
   STATUS[49].EXT.Maintanence := FALSE;
   STATUS[49].EXT.Operation := TRUE;
   STATUS[49].EXT.Forced := FALSE;
   STATUS[49].EXT.BIT29 := FALSE;
   STATUS[49].EXT.BIT30 := FALSE;
   STATUS[49].EXT.BIT31 := FALSE;
   STATUS[49].EXT.ModeBit1 := FALSE;
   STATUS[49].EXT.ModeBit2 := FALSE;
   STATUS[49].EXT.ModeBit3 := FALSE;
   STATUS[49].EXT.BIT19 := FALSE;
   STATUS[49].EXT.BIT20 := FALSE;
   STATUS[49].EXT.AlarmSuppressed := TRUE;
   STATUS[49].EXT.AlarmPrsent := FALSE;
   STATUS[49].EXT.AlarmFailUnAck := FALSE;
   STATUS[49].Status := 1;
   STATUS[49].TimeStamp := 16#3928;
   STATUS[50].VALUE := -11.85185;
   STATUS[50].TRIGVALUE := -11.85185;
   STATUS[50].EXT.AlarmWarnUnAck := FALSE;
   STATUS[50].EXT.AckRequired := FALSE;
   STATUS[50].EXT.Maintanence := FALSE;
   STATUS[50].EXT.Operation := TRUE;
   STATUS[50].EXT.Forced := FALSE;
   STATUS[50].EXT.BIT29 := FALSE;
   STATUS[50].EXT.BIT30 := FALSE;
   STATUS[50].EXT.BIT31 := FALSE;
   STATUS[50].EXT.ModeBit1 := FALSE;
   STATUS[50].EXT.ModeBit2 := FALSE;
   STATUS[50].EXT.ModeBit3 := FALSE;
   STATUS[50].EXT.BIT19 := FALSE;
   STATUS[50].EXT.BIT20 := FALSE;
   STATUS[50].EXT.AlarmSuppressed := TRUE;
   STATUS[50].EXT.AlarmPrsent := TRUE;
   STATUS[50].EXT.AlarmFailUnAck := TRUE;
   STATUS[50].Status := 150;
   STATUS[50].TimeStamp := 16#9344;
   STATUS[51].VALUE := -11.85185;
   STATUS[51].TRIGVALUE := -11.85185;
   STATUS[51].EXT.AlarmWarnUnAck := FALSE;
   STATUS[51].EXT.AckRequired := FALSE;
   STATUS[51].EXT.Maintanence := FALSE;
   STATUS[51].EXT.Operation := TRUE;
   STATUS[51].EXT.Forced := FALSE;
   STATUS[51].EXT.BIT29 := FALSE;
   STATUS[51].EXT.BIT30 := FALSE;
   STATUS[51].EXT.BIT31 := FALSE;
   STATUS[51].EXT.ModeBit1 := FALSE;
   STATUS[51].EXT.ModeBit2 := FALSE;
   STATUS[51].EXT.ModeBit3 := FALSE;
   STATUS[51].EXT.BIT19 := FALSE;
   STATUS[51].EXT.BIT20 := FALSE;
   STATUS[51].EXT.AlarmSuppressed := TRUE;
   STATUS[51].EXT.AlarmPrsent := TRUE;
   STATUS[51].EXT.AlarmFailUnAck := TRUE;
   STATUS[51].Status := 150;
   STATUS[51].TimeStamp := 16#9344;
   STATUS[52].VALUE := 0.0;
   STATUS[52].TRIGVALUE := 0.0;
   STATUS[52].EXT.AlarmWarnUnAck := TRUE;
   STATUS[52].EXT.AckRequired := FALSE;
   STATUS[52].EXT.Maintanence := FALSE;
   STATUS[52].EXT.Operation := TRUE;
   STATUS[52].EXT.Forced := FALSE;
   STATUS[52].EXT.BIT29 := FALSE;
   STATUS[52].EXT.BIT30 := FALSE;
   STATUS[52].EXT.BIT31 := FALSE;
   STATUS[52].EXT.ModeBit1 := FALSE;
   STATUS[52].EXT.ModeBit2 := FALSE;
   STATUS[52].EXT.ModeBit3 := FALSE;
   STATUS[52].EXT.BIT19 := FALSE;
   STATUS[52].EXT.BIT20 := FALSE;
   STATUS[52].EXT.AlarmSuppressed := TRUE;
   STATUS[52].EXT.AlarmPrsent := FALSE;
   STATUS[52].EXT.AlarmFailUnAck := FALSE;
   STATUS[52].Status := 1;
   STATUS[52].TimeStamp := 16#3928;
   STATUS[53].VALUE := 7.625868;
   STATUS[53].TRIGVALUE := 0.0;
   STATUS[53].EXT.AlarmWarnUnAck := TRUE;
   STATUS[53].EXT.AckRequired := FALSE;
   STATUS[53].EXT.Maintanence := FALSE;
   STATUS[53].EXT.Operation := TRUE;
   STATUS[53].EXT.Forced := FALSE;
   STATUS[53].EXT.BIT29 := FALSE;
   STATUS[53].EXT.BIT30 := FALSE;
   STATUS[53].EXT.BIT31 := FALSE;
   STATUS[53].EXT.ModeBit1 := FALSE;
   STATUS[53].EXT.ModeBit2 := FALSE;
   STATUS[53].EXT.ModeBit3 := FALSE;
   STATUS[53].EXT.BIT19 := FALSE;
   STATUS[53].EXT.BIT20 := FALSE;
   STATUS[53].EXT.AlarmSuppressed := TRUE;
   STATUS[53].EXT.AlarmPrsent := FALSE;
   STATUS[53].EXT.AlarmFailUnAck := FALSE;
   STATUS[53].Status := 1;
   STATUS[53].TimeStamp := 16#3928;
   STATUS[54].VALUE := 69.60178;
   STATUS[54].TRIGVALUE := 0.0;
   STATUS[54].EXT.AlarmWarnUnAck := TRUE;
   STATUS[54].EXT.AckRequired := FALSE;
   STATUS[54].EXT.Maintanence := FALSE;
   STATUS[54].EXT.Operation := TRUE;
   STATUS[54].EXT.Forced := FALSE;
   STATUS[54].EXT.BIT29 := FALSE;
   STATUS[54].EXT.BIT30 := FALSE;
   STATUS[54].EXT.BIT31 := FALSE;
   STATUS[54].EXT.ModeBit1 := FALSE;
   STATUS[54].EXT.ModeBit2 := FALSE;
   STATUS[54].EXT.ModeBit3 := FALSE;
   STATUS[54].EXT.BIT19 := FALSE;
   STATUS[54].EXT.BIT20 := FALSE;
   STATUS[54].EXT.AlarmSuppressed := TRUE;
   STATUS[54].EXT.AlarmPrsent := FALSE;
   STATUS[54].EXT.AlarmFailUnAck := FALSE;
   STATUS[54].Status := 1;
   STATUS[54].TimeStamp := 16#3928;
   STATUS[55].VALUE := -11.85185;
   STATUS[55].TRIGVALUE := -11.85185;
   STATUS[55].EXT.AlarmWarnUnAck := FALSE;
   STATUS[55].EXT.AckRequired := FALSE;
   STATUS[55].EXT.Maintanence := FALSE;
   STATUS[55].EXT.Operation := TRUE;
   STATUS[55].EXT.Forced := FALSE;
   STATUS[55].EXT.BIT29 := FALSE;
   STATUS[55].EXT.BIT30 := FALSE;
   STATUS[55].EXT.BIT31 := FALSE;
   STATUS[55].EXT.ModeBit1 := FALSE;
   STATUS[55].EXT.ModeBit2 := FALSE;
   STATUS[55].EXT.ModeBit3 := FALSE;
   STATUS[55].EXT.BIT19 := FALSE;
   STATUS[55].EXT.BIT20 := FALSE;
   STATUS[55].EXT.AlarmSuppressed := TRUE;
   STATUS[55].EXT.AlarmPrsent := TRUE;
   STATUS[55].EXT.AlarmFailUnAck := TRUE;
   STATUS[55].Status := 150;
   STATUS[55].TimeStamp := 16#9344;
   STATUS[56].VALUE := 0.0;
   STATUS[56].TRIGVALUE := 0.0;
   STATUS[56].EXT.AlarmWarnUnAck := TRUE;
   STATUS[56].EXT.AckRequired := FALSE;
   STATUS[56].EXT.Maintanence := FALSE;
   STATUS[56].EXT.Operation := TRUE;
   STATUS[56].EXT.Forced := FALSE;
   STATUS[56].EXT.BIT29 := FALSE;
   STATUS[56].EXT.BIT30 := FALSE;
   STATUS[56].EXT.BIT31 := FALSE;
   STATUS[56].EXT.ModeBit1 := FALSE;
   STATUS[56].EXT.ModeBit2 := FALSE;
   STATUS[56].EXT.ModeBit3 := FALSE;
   STATUS[56].EXT.BIT19 := FALSE;
   STATUS[56].EXT.BIT20 := FALSE;
   STATUS[56].EXT.AlarmSuppressed := TRUE;
   STATUS[56].EXT.AlarmPrsent := FALSE;
   STATUS[56].EXT.AlarmFailUnAck := FALSE;
   STATUS[56].Status := 1;
   STATUS[56].TimeStamp := 16#3928;
   STATUS[57].VALUE := 0.0;
   STATUS[57].TRIGVALUE := 0.0;
   STATUS[57].EXT.AlarmWarnUnAck := TRUE;
   STATUS[57].EXT.AckRequired := FALSE;
   STATUS[57].EXT.Maintanence := FALSE;
   STATUS[57].EXT.Operation := TRUE;
   STATUS[57].EXT.Forced := FALSE;
   STATUS[57].EXT.BIT29 := FALSE;
   STATUS[57].EXT.BIT30 := FALSE;
   STATUS[57].EXT.BIT31 := FALSE;
   STATUS[57].EXT.ModeBit1 := FALSE;
   STATUS[57].EXT.ModeBit2 := FALSE;
   STATUS[57].EXT.ModeBit3 := FALSE;
   STATUS[57].EXT.BIT19 := FALSE;
   STATUS[57].EXT.BIT20 := FALSE;
   STATUS[57].EXT.AlarmSuppressed := TRUE;
   STATUS[57].EXT.AlarmPrsent := FALSE;
   STATUS[57].EXT.AlarmFailUnAck := FALSE;
   STATUS[57].Status := 1;
   STATUS[57].TimeStamp := 16#3928;
   STATUS[58].VALUE := -11.85185;
   STATUS[58].TRIGVALUE := -11.85185;
   STATUS[58].EXT.AlarmWarnUnAck := FALSE;
   STATUS[58].EXT.AckRequired := FALSE;
   STATUS[58].EXT.Maintanence := FALSE;
   STATUS[58].EXT.Operation := TRUE;
   STATUS[58].EXT.Forced := FALSE;
   STATUS[58].EXT.BIT29 := FALSE;
   STATUS[58].EXT.BIT30 := FALSE;
   STATUS[58].EXT.BIT31 := FALSE;
   STATUS[58].EXT.ModeBit1 := FALSE;
   STATUS[58].EXT.ModeBit2 := FALSE;
   STATUS[58].EXT.ModeBit3 := FALSE;
   STATUS[58].EXT.BIT19 := FALSE;
   STATUS[58].EXT.BIT20 := FALSE;
   STATUS[58].EXT.AlarmSuppressed := TRUE;
   STATUS[58].EXT.AlarmPrsent := TRUE;
   STATUS[58].EXT.AlarmFailUnAck := TRUE;
   STATUS[58].Status := 150;
   STATUS[58].TimeStamp := 16#9344;
   STATUS[59].VALUE := 8.648004;
   STATUS[59].TRIGVALUE := 9.953704;
   STATUS[59].EXT.AlarmWarnUnAck := FALSE;
   STATUS[59].EXT.AckRequired := FALSE;
   STATUS[59].EXT.Maintanence := FALSE;
   STATUS[59].EXT.Operation := TRUE;
   STATUS[59].EXT.Forced := FALSE;
   STATUS[59].EXT.BIT29 := FALSE;
   STATUS[59].EXT.BIT30 := FALSE;
   STATUS[59].EXT.BIT31 := FALSE;
   STATUS[59].EXT.ModeBit1 := FALSE;
   STATUS[59].EXT.ModeBit2 := FALSE;
   STATUS[59].EXT.ModeBit3 := FALSE;
   STATUS[59].EXT.BIT19 := FALSE;
   STATUS[59].EXT.BIT20 := FALSE;
   STATUS[59].EXT.AlarmSuppressed := TRUE;
   STATUS[59].EXT.AlarmPrsent := TRUE;
   STATUS[59].EXT.AlarmFailUnAck := TRUE;
   STATUS[59].Status := 176;
   STATUS[59].TimeStamp := 16#C55A;
   STATUS[60].VALUE := -11.85185;
   STATUS[60].TRIGVALUE := -11.85185;
   STATUS[60].EXT.AlarmWarnUnAck := FALSE;
   STATUS[60].EXT.AckRequired := FALSE;
   STATUS[60].EXT.Maintanence := FALSE;
   STATUS[60].EXT.Operation := TRUE;
   STATUS[60].EXT.Forced := FALSE;
   STATUS[60].EXT.BIT29 := FALSE;
   STATUS[60].EXT.BIT30 := FALSE;
   STATUS[60].EXT.BIT31 := FALSE;
   STATUS[60].EXT.ModeBit1 := FALSE;
   STATUS[60].EXT.ModeBit2 := FALSE;
   STATUS[60].EXT.ModeBit3 := FALSE;
   STATUS[60].EXT.BIT19 := FALSE;
   STATUS[60].EXT.BIT20 := FALSE;
   STATUS[60].EXT.AlarmSuppressed := TRUE;
   STATUS[60].EXT.AlarmPrsent := TRUE;
   STATUS[60].EXT.AlarmFailUnAck := TRUE;
   STATUS[60].Status := 150;
   STATUS[60].TimeStamp := 16#9344;
   STATUS[61].VALUE := 118.5149;
   STATUS[61].TRIGVALUE := 118.5149;
   STATUS[61].EXT.AlarmWarnUnAck := FALSE;
   STATUS[61].EXT.AckRequired := FALSE;
   STATUS[61].EXT.Maintanence := FALSE;
   STATUS[61].EXT.Operation := TRUE;
   STATUS[61].EXT.Forced := FALSE;
   STATUS[61].EXT.BIT29 := FALSE;
   STATUS[61].EXT.BIT30 := FALSE;
   STATUS[61].EXT.BIT31 := FALSE;
   STATUS[61].EXT.ModeBit1 := FALSE;
   STATUS[61].EXT.ModeBit2 := FALSE;
   STATUS[61].EXT.ModeBit3 := FALSE;
   STATUS[61].EXT.BIT19 := FALSE;
   STATUS[61].EXT.BIT20 := FALSE;
   STATUS[61].EXT.AlarmSuppressed := TRUE;
   STATUS[61].EXT.AlarmPrsent := TRUE;
   STATUS[61].EXT.AlarmFailUnAck := TRUE;
   STATUS[61].Status := 151;
   STATUS[61].TimeStamp := 16#6499;
   STATUS[62].VALUE := 16.59209;
   STATUS[62].TRIGVALUE := 16.59209;
   STATUS[62].EXT.AlarmWarnUnAck := FALSE;
   STATUS[62].EXT.AckRequired := FALSE;
   STATUS[62].EXT.Maintanence := FALSE;
   STATUS[62].EXT.Operation := TRUE;
   STATUS[62].EXT.Forced := FALSE;
   STATUS[62].EXT.BIT29 := FALSE;
   STATUS[62].EXT.BIT30 := FALSE;
   STATUS[62].EXT.BIT31 := FALSE;
   STATUS[62].EXT.ModeBit1 := FALSE;
   STATUS[62].EXT.ModeBit2 := FALSE;
   STATUS[62].EXT.ModeBit3 := FALSE;
   STATUS[62].EXT.BIT19 := FALSE;
   STATUS[62].EXT.BIT20 := FALSE;
   STATUS[62].EXT.AlarmSuppressed := TRUE;
   STATUS[62].EXT.AlarmPrsent := TRUE;
   STATUS[62].EXT.AlarmFailUnAck := TRUE;
   STATUS[62].Status := 151;
   STATUS[62].TimeStamp := 16#9344;
   STATUS[63].VALUE := 118.5149;
   STATUS[63].TRIGVALUE := 118.5149;
   STATUS[63].EXT.AlarmWarnUnAck := FALSE;
   STATUS[63].EXT.AckRequired := FALSE;
   STATUS[63].EXT.Maintanence := FALSE;
   STATUS[63].EXT.Operation := TRUE;
   STATUS[63].EXT.Forced := FALSE;
   STATUS[63].EXT.BIT29 := FALSE;
   STATUS[63].EXT.BIT30 := FALSE;
   STATUS[63].EXT.BIT31 := FALSE;
   STATUS[63].EXT.ModeBit1 := FALSE;
   STATUS[63].EXT.ModeBit2 := FALSE;
   STATUS[63].EXT.ModeBit3 := FALSE;
   STATUS[63].EXT.BIT19 := FALSE;
   STATUS[63].EXT.BIT20 := FALSE;
   STATUS[63].EXT.AlarmSuppressed := FALSE;
   STATUS[63].EXT.AlarmPrsent := TRUE;
   STATUS[63].EXT.AlarmFailUnAck := TRUE;
   STATUS[63].Status := 151;
   STATUS[63].TimeStamp := 16#9344;
   STATUS[64].VALUE := -118.5185;
   STATUS[64].TRIGVALUE := -118.5185;
   STATUS[64].EXT.AlarmWarnUnAck := FALSE;
   STATUS[64].EXT.AckRequired := FALSE;
   STATUS[64].EXT.Maintanence := FALSE;
   STATUS[64].EXT.Operation := TRUE;
   STATUS[64].EXT.Forced := FALSE;
   STATUS[64].EXT.BIT29 := FALSE;
   STATUS[64].EXT.BIT30 := FALSE;
   STATUS[64].EXT.BIT31 := FALSE;
   STATUS[64].EXT.ModeBit1 := FALSE;
   STATUS[64].EXT.ModeBit2 := FALSE;
   STATUS[64].EXT.ModeBit3 := FALSE;
   STATUS[64].EXT.BIT19 := FALSE;
   STATUS[64].EXT.BIT20 := FALSE;
   STATUS[64].EXT.AlarmSuppressed := FALSE;
   STATUS[64].EXT.AlarmPrsent := TRUE;
   STATUS[64].EXT.AlarmFailUnAck := TRUE;
   STATUS[64].Status := 150;
   STATUS[64].TimeStamp := 16#8CA0;
   STATUS[65].VALUE := 118.5149;
   STATUS[65].TRIGVALUE := 118.5149;
   STATUS[65].EXT.AlarmWarnUnAck := FALSE;
   STATUS[65].EXT.AckRequired := FALSE;
   STATUS[65].EXT.Maintanence := FALSE;
   STATUS[65].EXT.Operation := TRUE;
   STATUS[65].EXT.Forced := FALSE;
   STATUS[65].EXT.BIT29 := FALSE;
   STATUS[65].EXT.BIT30 := FALSE;
   STATUS[65].EXT.BIT31 := FALSE;
   STATUS[65].EXT.ModeBit1 := FALSE;
   STATUS[65].EXT.ModeBit2 := FALSE;
   STATUS[65].EXT.ModeBit3 := FALSE;
   STATUS[65].EXT.BIT19 := FALSE;
   STATUS[65].EXT.BIT20 := FALSE;
   STATUS[65].EXT.AlarmSuppressed := TRUE;
   STATUS[65].EXT.AlarmPrsent := TRUE;
   STATUS[65].EXT.AlarmFailUnAck := TRUE;
   STATUS[65].Status := 151;
   STATUS[65].TimeStamp := 16#8CA0;
   STATUS[66].VALUE := 16.59209;
   STATUS[66].TRIGVALUE := 16.59209;
   STATUS[66].EXT.AlarmWarnUnAck := FALSE;
   STATUS[66].EXT.AckRequired := FALSE;
   STATUS[66].EXT.Maintanence := FALSE;
   STATUS[66].EXT.Operation := TRUE;
   STATUS[66].EXT.Forced := FALSE;
   STATUS[66].EXT.BIT29 := FALSE;
   STATUS[66].EXT.BIT30 := FALSE;
   STATUS[66].EXT.BIT31 := FALSE;
   STATUS[66].EXT.ModeBit1 := FALSE;
   STATUS[66].EXT.ModeBit2 := FALSE;
   STATUS[66].EXT.ModeBit3 := FALSE;
   STATUS[66].EXT.BIT19 := FALSE;
   STATUS[66].EXT.BIT20 := FALSE;
   STATUS[66].EXT.AlarmSuppressed := TRUE;
   STATUS[66].EXT.AlarmPrsent := TRUE;
   STATUS[66].EXT.AlarmFailUnAck := TRUE;
   STATUS[66].Status := 151;
   STATUS[66].TimeStamp := 16#9344;
   STATUS[67].VALUE := 1218.587;
   STATUS[67].TRIGVALUE := 115.1801;
   STATUS[67].EXT.AlarmWarnUnAck := TRUE;
   STATUS[67].EXT.AckRequired := FALSE;
   STATUS[67].EXT.Maintanence := FALSE;
   STATUS[67].EXT.Operation := TRUE;
   STATUS[67].EXT.Forced := FALSE;
   STATUS[67].EXT.BIT29 := FALSE;
   STATUS[67].EXT.BIT30 := FALSE;
   STATUS[67].EXT.BIT31 := FALSE;
   STATUS[67].EXT.ModeBit1 := FALSE;
   STATUS[67].EXT.ModeBit2 := FALSE;
   STATUS[67].EXT.ModeBit3 := FALSE;
   STATUS[67].EXT.BIT19 := FALSE;
   STATUS[67].EXT.BIT20 := FALSE;
   STATUS[67].EXT.AlarmSuppressed := TRUE;
   STATUS[67].EXT.AlarmPrsent := FALSE;
   STATUS[67].EXT.AlarmFailUnAck := FALSE;
   STATUS[67].Status := 1;
   STATUS[67].TimeStamp := 16#B806;
   STATUS[68].VALUE := 3.934896;
   STATUS[68].TRIGVALUE := 2.023438;
   STATUS[68].EXT.AlarmWarnUnAck := TRUE;
   STATUS[68].EXT.AckRequired := FALSE;
   STATUS[68].EXT.Maintanence := FALSE;
   STATUS[68].EXT.Operation := TRUE;
   STATUS[68].EXT.Forced := FALSE;
   STATUS[68].EXT.BIT29 := FALSE;
   STATUS[68].EXT.BIT30 := FALSE;
   STATUS[68].EXT.BIT31 := FALSE;
   STATUS[68].EXT.ModeBit1 := FALSE;
   STATUS[68].EXT.ModeBit2 := FALSE;
   STATUS[68].EXT.ModeBit3 := FALSE;
   STATUS[68].EXT.BIT19 := FALSE;
   STATUS[68].EXT.BIT20 := FALSE;
   STATUS[68].EXT.AlarmSuppressed := TRUE;
   STATUS[68].EXT.AlarmPrsent := FALSE;
   STATUS[68].EXT.AlarmFailUnAck := FALSE;
   STATUS[68].Status := 1;
   STATUS[68].TimeStamp := 16#B800;
   STATUS[69].VALUE := 1183.648;
   STATUS[69].TRIGVALUE := 148.3833;
   STATUS[69].EXT.AlarmWarnUnAck := TRUE;
   STATUS[69].EXT.AckRequired := FALSE;
   STATUS[69].EXT.Maintanence := FALSE;
   STATUS[69].EXT.Operation := TRUE;
   STATUS[69].EXT.Forced := FALSE;
   STATUS[69].EXT.BIT29 := FALSE;
   STATUS[69].EXT.BIT30 := FALSE;
   STATUS[69].EXT.BIT31 := FALSE;
   STATUS[69].EXT.ModeBit1 := FALSE;
   STATUS[69].EXT.ModeBit2 := FALSE;
   STATUS[69].EXT.ModeBit3 := FALSE;
   STATUS[69].EXT.BIT19 := FALSE;
   STATUS[69].EXT.BIT20 := FALSE;
   STATUS[69].EXT.AlarmSuppressed := TRUE;
   STATUS[69].EXT.AlarmPrsent := FALSE;
   STATUS[69].EXT.AlarmFailUnAck := FALSE;
   STATUS[69].Status := 1;
   STATUS[69].TimeStamp := 16#A991;
   STATUS[70].VALUE := 3.875651;
   STATUS[70].TRIGVALUE := 1.142253;
   STATUS[70].EXT.AlarmWarnUnAck := TRUE;
   STATUS[70].EXT.AckRequired := FALSE;
   STATUS[70].EXT.Maintanence := FALSE;
   STATUS[70].EXT.Operation := TRUE;
   STATUS[70].EXT.Forced := FALSE;
   STATUS[70].EXT.BIT29 := FALSE;
   STATUS[70].EXT.BIT30 := FALSE;
   STATUS[70].EXT.BIT31 := FALSE;
   STATUS[70].EXT.ModeBit1 := FALSE;
   STATUS[70].EXT.ModeBit2 := FALSE;
   STATUS[70].EXT.ModeBit3 := FALSE;
   STATUS[70].EXT.BIT19 := FALSE;
   STATUS[70].EXT.BIT20 := FALSE;
   STATUS[70].EXT.AlarmSuppressed := TRUE;
   STATUS[70].EXT.AlarmPrsent := FALSE;
   STATUS[70].EXT.AlarmFailUnAck := FALSE;
   STATUS[70].Status := 1;
   STATUS[70].TimeStamp := 16#A95B;
   STATUS[71].VALUE := 1355.469;
   STATUS[71].TRIGVALUE := 158.5829;
   STATUS[71].EXT.AlarmWarnUnAck := TRUE;
   STATUS[71].EXT.AckRequired := FALSE;
   STATUS[71].EXT.Maintanence := FALSE;
   STATUS[71].EXT.Operation := TRUE;
   STATUS[71].EXT.Forced := FALSE;
   STATUS[71].EXT.BIT29 := FALSE;
   STATUS[71].EXT.BIT30 := FALSE;
   STATUS[71].EXT.BIT31 := FALSE;
   STATUS[71].EXT.ModeBit1 := FALSE;
   STATUS[71].EXT.ModeBit2 := FALSE;
   STATUS[71].EXT.ModeBit3 := FALSE;
   STATUS[71].EXT.BIT19 := FALSE;
   STATUS[71].EXT.BIT20 := FALSE;
   STATUS[71].EXT.AlarmSuppressed := TRUE;
   STATUS[71].EXT.AlarmPrsent := FALSE;
   STATUS[71].EXT.AlarmFailUnAck := FALSE;
   STATUS[71].Status := 1;
   STATUS[71].TimeStamp := 16#0020;
   STATUS[72].VALUE := 4.802734;
   STATUS[72].TRIGVALUE := 1.56543;
   STATUS[72].EXT.AlarmWarnUnAck := TRUE;
   STATUS[72].EXT.AckRequired := FALSE;
   STATUS[72].EXT.Maintanence := FALSE;
   STATUS[72].EXT.Operation := TRUE;
   STATUS[72].EXT.Forced := FALSE;
   STATUS[72].EXT.BIT29 := FALSE;
   STATUS[72].EXT.BIT30 := FALSE;
   STATUS[72].EXT.BIT31 := FALSE;
   STATUS[72].EXT.ModeBit1 := FALSE;
   STATUS[72].EXT.ModeBit2 := FALSE;
   STATUS[72].EXT.ModeBit3 := FALSE;
   STATUS[72].EXT.BIT19 := FALSE;
   STATUS[72].EXT.BIT20 := FALSE;
   STATUS[72].EXT.AlarmSuppressed := TRUE;
   STATUS[72].EXT.AlarmPrsent := FALSE;
   STATUS[72].EXT.AlarmFailUnAck := FALSE;
   STATUS[72].Status := 1;
   STATUS[72].TimeStamp := 16#EA4A;
   STATUS[73].VALUE := 1296.984;
   STATUS[73].TRIGVALUE := 141.3845;
   STATUS[73].EXT.AlarmWarnUnAck := TRUE;
   STATUS[73].EXT.AckRequired := FALSE;
   STATUS[73].EXT.Maintanence := FALSE;
   STATUS[73].EXT.Operation := TRUE;
   STATUS[73].EXT.Forced := FALSE;
   STATUS[73].EXT.BIT29 := FALSE;
   STATUS[73].EXT.BIT30 := FALSE;
   STATUS[73].EXT.BIT31 := FALSE;
   STATUS[73].EXT.ModeBit1 := FALSE;
   STATUS[73].EXT.ModeBit2 := FALSE;
   STATUS[73].EXT.ModeBit3 := FALSE;
   STATUS[73].EXT.BIT19 := FALSE;
   STATUS[73].EXT.BIT20 := FALSE;
   STATUS[73].EXT.AlarmSuppressed := TRUE;
   STATUS[73].EXT.AlarmPrsent := FALSE;
   STATUS[73].EXT.AlarmFailUnAck := FALSE;
   STATUS[73].Status := 1;
   STATUS[73].TimeStamp := 16#6B5A;
   STATUS[74].VALUE := 4.843424;
   STATUS[74].TRIGVALUE := 1.541992;
   STATUS[74].EXT.AlarmWarnUnAck := TRUE;
   STATUS[74].EXT.AckRequired := FALSE;
   STATUS[74].EXT.Maintanence := FALSE;
   STATUS[74].EXT.Operation := TRUE;
   STATUS[74].EXT.Forced := FALSE;
   STATUS[74].EXT.BIT29 := FALSE;
   STATUS[74].EXT.BIT30 := FALSE;
   STATUS[74].EXT.BIT31 := FALSE;
   STATUS[74].EXT.ModeBit1 := FALSE;
   STATUS[74].EXT.ModeBit2 := FALSE;
   STATUS[74].EXT.ModeBit3 := FALSE;
   STATUS[74].EXT.BIT19 := FALSE;
   STATUS[74].EXT.BIT20 := FALSE;
   STATUS[74].EXT.AlarmSuppressed := TRUE;
   STATUS[74].EXT.AlarmPrsent := FALSE;
   STATUS[74].EXT.AlarmFailUnAck := FALSE;
   STATUS[74].Status := 1;
   STATUS[74].TimeStamp := 16#E14B;
   STATUS[75].VALUE := -1777.778;
   STATUS[75].TRIGVALUE := -1777.778;
   STATUS[75].EXT.AlarmWarnUnAck := FALSE;
   STATUS[75].EXT.AckRequired := FALSE;
   STATUS[75].EXT.Maintanence := FALSE;
   STATUS[75].EXT.Operation := TRUE;
   STATUS[75].EXT.Forced := FALSE;
   STATUS[75].EXT.BIT29 := FALSE;
   STATUS[75].EXT.BIT30 := FALSE;
   STATUS[75].EXT.BIT31 := FALSE;
   STATUS[75].EXT.ModeBit1 := FALSE;
   STATUS[75].EXT.ModeBit2 := FALSE;
   STATUS[75].EXT.ModeBit3 := FALSE;
   STATUS[75].EXT.BIT19 := FALSE;
   STATUS[75].EXT.BIT20 := FALSE;
   STATUS[75].EXT.AlarmSuppressed := TRUE;
   STATUS[75].EXT.AlarmPrsent := TRUE;
   STATUS[75].EXT.AlarmFailUnAck := TRUE;
   STATUS[75].Status := 150;
   STATUS[75].TimeStamp := 16#9344;
   STATUS[76].VALUE := -10.66667;
   STATUS[76].TRIGVALUE := -10.66667;
   STATUS[76].EXT.AlarmWarnUnAck := FALSE;
   STATUS[76].EXT.AckRequired := FALSE;
   STATUS[76].EXT.Maintanence := FALSE;
   STATUS[76].EXT.Operation := TRUE;
   STATUS[76].EXT.Forced := FALSE;
   STATUS[76].EXT.BIT29 := FALSE;
   STATUS[76].EXT.BIT30 := FALSE;
   STATUS[76].EXT.BIT31 := FALSE;
   STATUS[76].EXT.ModeBit1 := FALSE;
   STATUS[76].EXT.ModeBit2 := FALSE;
   STATUS[76].EXT.ModeBit3 := FALSE;
   STATUS[76].EXT.BIT19 := FALSE;
   STATUS[76].EXT.BIT20 := FALSE;
   STATUS[76].EXT.AlarmSuppressed := TRUE;
   STATUS[76].EXT.AlarmPrsent := TRUE;
   STATUS[76].EXT.AlarmFailUnAck := TRUE;
   STATUS[76].Status := 150;
   STATUS[76].TimeStamp := 16#9344;
   STATUS[77].VALUE := -118.5185;
   STATUS[77].TRIGVALUE := -118.5185;
   STATUS[77].EXT.AlarmWarnUnAck := FALSE;
   STATUS[77].EXT.AckRequired := FALSE;
   STATUS[77].EXT.Maintanence := FALSE;
   STATUS[77].EXT.Operation := TRUE;
   STATUS[77].EXT.Forced := FALSE;
   STATUS[77].EXT.BIT29 := FALSE;
   STATUS[77].EXT.BIT30 := FALSE;
   STATUS[77].EXT.BIT31 := FALSE;
   STATUS[77].EXT.ModeBit1 := FALSE;
   STATUS[77].EXT.ModeBit2 := FALSE;
   STATUS[77].EXT.ModeBit3 := FALSE;
   STATUS[77].EXT.BIT19 := FALSE;
   STATUS[77].EXT.BIT20 := FALSE;
   STATUS[77].EXT.AlarmSuppressed := TRUE;
   STATUS[77].EXT.AlarmPrsent := TRUE;
   STATUS[77].EXT.AlarmFailUnAck := TRUE;
   STATUS[77].Status := 150;
   STATUS[77].TimeStamp := 16#9344;
   STATUS[78].VALUE := 0.0;
   STATUS[78].TRIGVALUE := 0.0;
   STATUS[78].EXT.AlarmWarnUnAck := FALSE;
   STATUS[78].EXT.AckRequired := FALSE;
   STATUS[78].EXT.Maintanence := FALSE;
   STATUS[78].EXT.Operation := FALSE;
   STATUS[78].EXT.Forced := FALSE;
   STATUS[78].EXT.BIT29 := FALSE;
   STATUS[78].EXT.BIT30 := FALSE;
   STATUS[78].EXT.BIT31 := FALSE;
   STATUS[78].EXT.ModeBit1 := FALSE;
   STATUS[78].EXT.ModeBit2 := FALSE;
   STATUS[78].EXT.ModeBit3 := FALSE;
   STATUS[78].EXT.BIT19 := FALSE;
   STATUS[78].EXT.BIT20 := FALSE;
   STATUS[78].EXT.AlarmSuppressed := FALSE;
   STATUS[78].EXT.AlarmPrsent := FALSE;
   STATUS[78].EXT.AlarmFailUnAck := FALSE;
   STATUS[78].Status := 0;
   STATUS[78].TimeStamp := 16#0000;
   STATUS[79].VALUE := 0.0;
   STATUS[79].TRIGVALUE := 0.0;
   STATUS[79].EXT.AlarmWarnUnAck := FALSE;
   STATUS[79].EXT.AckRequired := FALSE;
   STATUS[79].EXT.Maintanence := FALSE;
   STATUS[79].EXT.Operation := FALSE;
   STATUS[79].EXT.Forced := FALSE;
   STATUS[79].EXT.BIT29 := FALSE;
   STATUS[79].EXT.BIT30 := FALSE;
   STATUS[79].EXT.BIT31 := FALSE;
   STATUS[79].EXT.ModeBit1 := FALSE;
   STATUS[79].EXT.ModeBit2 := FALSE;
   STATUS[79].EXT.ModeBit3 := FALSE;
   STATUS[79].EXT.BIT19 := FALSE;
   STATUS[79].EXT.BIT20 := FALSE;
   STATUS[79].EXT.AlarmSuppressed := FALSE;
   STATUS[79].EXT.AlarmPrsent := FALSE;
   STATUS[79].EXT.AlarmFailUnAck := FALSE;
   STATUS[79].Status := 0;
   STATUS[79].TimeStamp := 16#0000;
   STATUS[80].VALUE := 0.0;
   STATUS[80].TRIGVALUE := 0.0;
   STATUS[80].EXT.AlarmWarnUnAck := FALSE;
   STATUS[80].EXT.AckRequired := FALSE;
   STATUS[80].EXT.Maintanence := FALSE;
   STATUS[80].EXT.Operation := FALSE;
   STATUS[80].EXT.Forced := FALSE;
   STATUS[80].EXT.BIT29 := FALSE;
   STATUS[80].EXT.BIT30 := FALSE;
   STATUS[80].EXT.BIT31 := FALSE;
   STATUS[80].EXT.ModeBit1 := FALSE;
   STATUS[80].EXT.ModeBit2 := FALSE;
   STATUS[80].EXT.ModeBit3 := FALSE;
   STATUS[80].EXT.BIT19 := FALSE;
   STATUS[80].EXT.BIT20 := FALSE;
   STATUS[80].EXT.AlarmSuppressed := FALSE;
   STATUS[80].EXT.AlarmPrsent := FALSE;
   STATUS[80].EXT.AlarmFailUnAck := FALSE;
   STATUS[80].Status := 0;
   STATUS[80].TimeStamp := 16#0000;
   STATUS[81].VALUE := 0.0;
   STATUS[81].TRIGVALUE := 0.0;
   STATUS[81].EXT.AlarmWarnUnAck := FALSE;
   STATUS[81].EXT.AckRequired := FALSE;
   STATUS[81].EXT.Maintanence := FALSE;
   STATUS[81].EXT.Operation := FALSE;
   STATUS[81].EXT.Forced := FALSE;
   STATUS[81].EXT.BIT29 := FALSE;
   STATUS[81].EXT.BIT30 := FALSE;
   STATUS[81].EXT.BIT31 := FALSE;
   STATUS[81].EXT.ModeBit1 := FALSE;
   STATUS[81].EXT.ModeBit2 := FALSE;
   STATUS[81].EXT.ModeBit3 := FALSE;
   STATUS[81].EXT.BIT19 := FALSE;
   STATUS[81].EXT.BIT20 := FALSE;
   STATUS[81].EXT.AlarmSuppressed := FALSE;
   STATUS[81].EXT.AlarmPrsent := FALSE;
   STATUS[81].EXT.AlarmFailUnAck := FALSE;
   STATUS[81].Status := 0;
   STATUS[81].TimeStamp := 16#0000;
   STATUS[82].VALUE := 0.0;
   STATUS[82].TRIGVALUE := 0.0;
   STATUS[82].EXT.AlarmWarnUnAck := FALSE;
   STATUS[82].EXT.AckRequired := FALSE;
   STATUS[82].EXT.Maintanence := FALSE;
   STATUS[82].EXT.Operation := FALSE;
   STATUS[82].EXT.Forced := FALSE;
   STATUS[82].EXT.BIT29 := FALSE;
   STATUS[82].EXT.BIT30 := FALSE;
   STATUS[82].EXT.BIT31 := FALSE;
   STATUS[82].EXT.ModeBit1 := FALSE;
   STATUS[82].EXT.ModeBit2 := FALSE;
   STATUS[82].EXT.ModeBit3 := FALSE;
   STATUS[82].EXT.BIT19 := FALSE;
   STATUS[82].EXT.BIT20 := FALSE;
   STATUS[82].EXT.AlarmSuppressed := FALSE;
   STATUS[82].EXT.AlarmPrsent := FALSE;
   STATUS[82].EXT.AlarmFailUnAck := FALSE;
   STATUS[82].Status := 0;
   STATUS[82].TimeStamp := 16#0000;
   STATUS[83].VALUE := 0.0;
   STATUS[83].TRIGVALUE := 0.0;
   STATUS[83].EXT.AlarmWarnUnAck := FALSE;
   STATUS[83].EXT.AckRequired := FALSE;
   STATUS[83].EXT.Maintanence := FALSE;
   STATUS[83].EXT.Operation := FALSE;
   STATUS[83].EXT.Forced := FALSE;
   STATUS[83].EXT.BIT29 := FALSE;
   STATUS[83].EXT.BIT30 := FALSE;
   STATUS[83].EXT.BIT31 := FALSE;
   STATUS[83].EXT.ModeBit1 := FALSE;
   STATUS[83].EXT.ModeBit2 := FALSE;
   STATUS[83].EXT.ModeBit3 := FALSE;
   STATUS[83].EXT.BIT19 := FALSE;
   STATUS[83].EXT.BIT20 := FALSE;
   STATUS[83].EXT.AlarmSuppressed := FALSE;
   STATUS[83].EXT.AlarmPrsent := FALSE;
   STATUS[83].EXT.AlarmFailUnAck := FALSE;
   STATUS[83].Status := 0;
   STATUS[83].TimeStamp := 16#0000;
   STATUS[84].VALUE := 0.0;
   STATUS[84].TRIGVALUE := 0.0;
   STATUS[84].EXT.AlarmWarnUnAck := FALSE;
   STATUS[84].EXT.AckRequired := FALSE;
   STATUS[84].EXT.Maintanence := FALSE;
   STATUS[84].EXT.Operation := FALSE;
   STATUS[84].EXT.Forced := FALSE;
   STATUS[84].EXT.BIT29 := FALSE;
   STATUS[84].EXT.BIT30 := FALSE;
   STATUS[84].EXT.BIT31 := FALSE;
   STATUS[84].EXT.ModeBit1 := FALSE;
   STATUS[84].EXT.ModeBit2 := FALSE;
   STATUS[84].EXT.ModeBit3 := FALSE;
   STATUS[84].EXT.BIT19 := FALSE;
   STATUS[84].EXT.BIT20 := FALSE;
   STATUS[84].EXT.AlarmSuppressed := FALSE;
   STATUS[84].EXT.AlarmPrsent := FALSE;
   STATUS[84].EXT.AlarmFailUnAck := FALSE;
   STATUS[84].Status := 0;
   STATUS[84].TimeStamp := 16#0000;
   STATUS[85].VALUE := 0.0;
   STATUS[85].TRIGVALUE := 0.0;
   STATUS[85].EXT.AlarmWarnUnAck := FALSE;
   STATUS[85].EXT.AckRequired := FALSE;
   STATUS[85].EXT.Maintanence := FALSE;
   STATUS[85].EXT.Operation := FALSE;
   STATUS[85].EXT.Forced := FALSE;
   STATUS[85].EXT.BIT29 := FALSE;
   STATUS[85].EXT.BIT30 := FALSE;
   STATUS[85].EXT.BIT31 := FALSE;
   STATUS[85].EXT.ModeBit1 := FALSE;
   STATUS[85].EXT.ModeBit2 := FALSE;
   STATUS[85].EXT.ModeBit3 := FALSE;
   STATUS[85].EXT.BIT19 := FALSE;
   STATUS[85].EXT.BIT20 := FALSE;
   STATUS[85].EXT.AlarmSuppressed := FALSE;
   STATUS[85].EXT.AlarmPrsent := FALSE;
   STATUS[85].EXT.AlarmFailUnAck := FALSE;
   STATUS[85].Status := 0;
   STATUS[85].TimeStamp := 16#0000;
   STATUS[86].VALUE := 0.0;
   STATUS[86].TRIGVALUE := 0.0;
   STATUS[86].EXT.AlarmWarnUnAck := FALSE;
   STATUS[86].EXT.AckRequired := FALSE;
   STATUS[86].EXT.Maintanence := FALSE;
   STATUS[86].EXT.Operation := FALSE;
   STATUS[86].EXT.Forced := FALSE;
   STATUS[86].EXT.BIT29 := FALSE;
   STATUS[86].EXT.BIT30 := FALSE;
   STATUS[86].EXT.BIT31 := FALSE;
   STATUS[86].EXT.ModeBit1 := FALSE;
   STATUS[86].EXT.ModeBit2 := FALSE;
   STATUS[86].EXT.ModeBit3 := FALSE;
   STATUS[86].EXT.BIT19 := FALSE;
   STATUS[86].EXT.BIT20 := FALSE;
   STATUS[86].EXT.AlarmSuppressed := FALSE;
   STATUS[86].EXT.AlarmPrsent := FALSE;
   STATUS[86].EXT.AlarmFailUnAck := FALSE;
   STATUS[86].Status := 0;
   STATUS[86].TimeStamp := 16#0000;
   STATUS[87].VALUE := 0.0;
   STATUS[87].TRIGVALUE := 0.0;
   STATUS[87].EXT.AlarmWarnUnAck := FALSE;
   STATUS[87].EXT.AckRequired := FALSE;
   STATUS[87].EXT.Maintanence := FALSE;
   STATUS[87].EXT.Operation := FALSE;
   STATUS[87].EXT.Forced := FALSE;
   STATUS[87].EXT.BIT29 := FALSE;
   STATUS[87].EXT.BIT30 := FALSE;
   STATUS[87].EXT.BIT31 := FALSE;
   STATUS[87].EXT.ModeBit1 := FALSE;
   STATUS[87].EXT.ModeBit2 := FALSE;
   STATUS[87].EXT.ModeBit3 := FALSE;
   STATUS[87].EXT.BIT19 := FALSE;
   STATUS[87].EXT.BIT20 := FALSE;
   STATUS[87].EXT.AlarmSuppressed := FALSE;
   STATUS[87].EXT.AlarmPrsent := FALSE;
   STATUS[87].EXT.AlarmFailUnAck := FALSE;
   STATUS[87].Status := 0;
   STATUS[87].TimeStamp := 16#0000;
   STATUS[88].VALUE := 0.0;
   STATUS[88].TRIGVALUE := 0.0;
   STATUS[88].EXT.AlarmWarnUnAck := FALSE;
   STATUS[88].EXT.AckRequired := FALSE;
   STATUS[88].EXT.Maintanence := FALSE;
   STATUS[88].EXT.Operation := FALSE;
   STATUS[88].EXT.Forced := FALSE;
   STATUS[88].EXT.BIT29 := FALSE;
   STATUS[88].EXT.BIT30 := FALSE;
   STATUS[88].EXT.BIT31 := FALSE;
   STATUS[88].EXT.ModeBit1 := FALSE;
   STATUS[88].EXT.ModeBit2 := FALSE;
   STATUS[88].EXT.ModeBit3 := FALSE;
   STATUS[88].EXT.BIT19 := FALSE;
   STATUS[88].EXT.BIT20 := FALSE;
   STATUS[88].EXT.AlarmSuppressed := FALSE;
   STATUS[88].EXT.AlarmPrsent := FALSE;
   STATUS[88].EXT.AlarmFailUnAck := FALSE;
   STATUS[88].Status := 0;
   STATUS[88].TimeStamp := 16#0000;
   STATUS[89].VALUE := 0.0;
   STATUS[89].TRIGVALUE := 0.0;
   STATUS[89].EXT.AlarmWarnUnAck := FALSE;
   STATUS[89].EXT.AckRequired := FALSE;
   STATUS[89].EXT.Maintanence := FALSE;
   STATUS[89].EXT.Operation := FALSE;
   STATUS[89].EXT.Forced := FALSE;
   STATUS[89].EXT.BIT29 := FALSE;
   STATUS[89].EXT.BIT30 := FALSE;
   STATUS[89].EXT.BIT31 := FALSE;
   STATUS[89].EXT.ModeBit1 := FALSE;
   STATUS[89].EXT.ModeBit2 := FALSE;
   STATUS[89].EXT.ModeBit3 := FALSE;
   STATUS[89].EXT.BIT19 := FALSE;
   STATUS[89].EXT.BIT20 := FALSE;
   STATUS[89].EXT.AlarmSuppressed := FALSE;
   STATUS[89].EXT.AlarmPrsent := FALSE;
   STATUS[89].EXT.AlarmFailUnAck := FALSE;
   STATUS[89].Status := 0;
   STATUS[89].TimeStamp := 16#0000;
   STATUS[90].VALUE := 0.0;
   STATUS[90].TRIGVALUE := 0.0;
   STATUS[90].EXT.AlarmWarnUnAck := FALSE;
   STATUS[90].EXT.AckRequired := FALSE;
   STATUS[90].EXT.Maintanence := FALSE;
   STATUS[90].EXT.Operation := FALSE;
   STATUS[90].EXT.Forced := FALSE;
   STATUS[90].EXT.BIT29 := FALSE;
   STATUS[90].EXT.BIT30 := FALSE;
   STATUS[90].EXT.BIT31 := FALSE;
   STATUS[90].EXT.ModeBit1 := FALSE;
   STATUS[90].EXT.ModeBit2 := FALSE;
   STATUS[90].EXT.ModeBit3 := FALSE;
   STATUS[90].EXT.BIT19 := FALSE;
   STATUS[90].EXT.BIT20 := FALSE;
   STATUS[90].EXT.AlarmSuppressed := FALSE;
   STATUS[90].EXT.AlarmPrsent := FALSE;
   STATUS[90].EXT.AlarmFailUnAck := FALSE;
   STATUS[90].Status := 0;
   STATUS[90].TimeStamp := 16#0000;
   STATUS[91].VALUE := 0.0;
   STATUS[91].TRIGVALUE := 0.0;
   STATUS[91].EXT.AlarmWarnUnAck := FALSE;
   STATUS[91].EXT.AckRequired := FALSE;
   STATUS[91].EXT.Maintanence := FALSE;
   STATUS[91].EXT.Operation := FALSE;
   STATUS[91].EXT.Forced := FALSE;
   STATUS[91].EXT.BIT29 := FALSE;
   STATUS[91].EXT.BIT30 := FALSE;
   STATUS[91].EXT.BIT31 := FALSE;
   STATUS[91].EXT.ModeBit1 := FALSE;
   STATUS[91].EXT.ModeBit2 := FALSE;
   STATUS[91].EXT.ModeBit3 := FALSE;
   STATUS[91].EXT.BIT19 := FALSE;
   STATUS[91].EXT.BIT20 := FALSE;
   STATUS[91].EXT.AlarmSuppressed := FALSE;
   STATUS[91].EXT.AlarmPrsent := FALSE;
   STATUS[91].EXT.AlarmFailUnAck := FALSE;
   STATUS[91].Status := 0;
   STATUS[91].TimeStamp := 16#0000;
   STATUS[92].VALUE := 0.0;
   STATUS[92].TRIGVALUE := 0.0;
   STATUS[92].EXT.AlarmWarnUnAck := FALSE;
   STATUS[92].EXT.AckRequired := FALSE;
   STATUS[92].EXT.Maintanence := FALSE;
   STATUS[92].EXT.Operation := FALSE;
   STATUS[92].EXT.Forced := FALSE;
   STATUS[92].EXT.BIT29 := FALSE;
   STATUS[92].EXT.BIT30 := FALSE;
   STATUS[92].EXT.BIT31 := FALSE;
   STATUS[92].EXT.ModeBit1 := FALSE;
   STATUS[92].EXT.ModeBit2 := FALSE;
   STATUS[92].EXT.ModeBit3 := FALSE;
   STATUS[92].EXT.BIT19 := FALSE;
   STATUS[92].EXT.BIT20 := FALSE;
   STATUS[92].EXT.AlarmSuppressed := FALSE;
   STATUS[92].EXT.AlarmPrsent := FALSE;
   STATUS[92].EXT.AlarmFailUnAck := FALSE;
   STATUS[92].Status := 0;
   STATUS[92].TimeStamp := 16#0000;
   STATUS[93].VALUE := 0.0;
   STATUS[93].TRIGVALUE := 0.0;
   STATUS[93].EXT.AlarmWarnUnAck := FALSE;
   STATUS[93].EXT.AckRequired := FALSE;
   STATUS[93].EXT.Maintanence := FALSE;
   STATUS[93].EXT.Operation := FALSE;
   STATUS[93].EXT.Forced := FALSE;
   STATUS[93].EXT.BIT29 := FALSE;
   STATUS[93].EXT.BIT30 := FALSE;
   STATUS[93].EXT.BIT31 := FALSE;
   STATUS[93].EXT.ModeBit1 := FALSE;
   STATUS[93].EXT.ModeBit2 := FALSE;
   STATUS[93].EXT.ModeBit3 := FALSE;
   STATUS[93].EXT.BIT19 := FALSE;
   STATUS[93].EXT.BIT20 := FALSE;
   STATUS[93].EXT.AlarmSuppressed := FALSE;
   STATUS[93].EXT.AlarmPrsent := FALSE;
   STATUS[93].EXT.AlarmFailUnAck := FALSE;
   STATUS[93].Status := 0;
   STATUS[93].TimeStamp := 16#0000;
   STATUS[94].VALUE := 0.0;
   STATUS[94].TRIGVALUE := 0.0;
   STATUS[94].EXT.AlarmWarnUnAck := FALSE;
   STATUS[94].EXT.AckRequired := FALSE;
   STATUS[94].EXT.Maintanence := FALSE;
   STATUS[94].EXT.Operation := FALSE;
   STATUS[94].EXT.Forced := FALSE;
   STATUS[94].EXT.BIT29 := FALSE;
   STATUS[94].EXT.BIT30 := FALSE;
   STATUS[94].EXT.BIT31 := FALSE;
   STATUS[94].EXT.ModeBit1 := FALSE;
   STATUS[94].EXT.ModeBit2 := FALSE;
   STATUS[94].EXT.ModeBit3 := FALSE;
   STATUS[94].EXT.BIT19 := FALSE;
   STATUS[94].EXT.BIT20 := FALSE;
   STATUS[94].EXT.AlarmSuppressed := FALSE;
   STATUS[94].EXT.AlarmPrsent := FALSE;
   STATUS[94].EXT.AlarmFailUnAck := FALSE;
   STATUS[94].Status := 0;
   STATUS[94].TimeStamp := 16#0000;
   STATUS[95].VALUE := 0.0;
   STATUS[95].TRIGVALUE := 0.0;
   STATUS[95].EXT.AlarmWarnUnAck := FALSE;
   STATUS[95].EXT.AckRequired := FALSE;
   STATUS[95].EXT.Maintanence := FALSE;
   STATUS[95].EXT.Operation := FALSE;
   STATUS[95].EXT.Forced := FALSE;
   STATUS[95].EXT.BIT29 := FALSE;
   STATUS[95].EXT.BIT30 := FALSE;
   STATUS[95].EXT.BIT31 := FALSE;
   STATUS[95].EXT.ModeBit1 := FALSE;
   STATUS[95].EXT.ModeBit2 := FALSE;
   STATUS[95].EXT.ModeBit3 := FALSE;
   STATUS[95].EXT.BIT19 := FALSE;
   STATUS[95].EXT.BIT20 := FALSE;
   STATUS[95].EXT.AlarmSuppressed := FALSE;
   STATUS[95].EXT.AlarmPrsent := FALSE;
   STATUS[95].EXT.AlarmFailUnAck := FALSE;
   STATUS[95].Status := 0;
   STATUS[95].TimeStamp := 16#0000;
   STATUS[96].VALUE := 0.0;
   STATUS[96].TRIGVALUE := 0.0;
   STATUS[96].EXT.AlarmWarnUnAck := FALSE;
   STATUS[96].EXT.AckRequired := FALSE;
   STATUS[96].EXT.Maintanence := FALSE;
   STATUS[96].EXT.Operation := FALSE;
   STATUS[96].EXT.Forced := FALSE;
   STATUS[96].EXT.BIT29 := FALSE;
   STATUS[96].EXT.BIT30 := FALSE;
   STATUS[96].EXT.BIT31 := FALSE;
   STATUS[96].EXT.ModeBit1 := FALSE;
   STATUS[96].EXT.ModeBit2 := FALSE;
   STATUS[96].EXT.ModeBit3 := FALSE;
   STATUS[96].EXT.BIT19 := FALSE;
   STATUS[96].EXT.BIT20 := FALSE;
   STATUS[96].EXT.AlarmSuppressed := FALSE;
   STATUS[96].EXT.AlarmPrsent := FALSE;
   STATUS[96].EXT.AlarmFailUnAck := FALSE;
   STATUS[96].Status := 0;
   STATUS[96].TimeStamp := 16#0000;
   STATUS[97].VALUE := 0.0;
   STATUS[97].TRIGVALUE := 0.0;
   STATUS[97].EXT.AlarmWarnUnAck := FALSE;
   STATUS[97].EXT.AckRequired := FALSE;
   STATUS[97].EXT.Maintanence := FALSE;
   STATUS[97].EXT.Operation := FALSE;
   STATUS[97].EXT.Forced := FALSE;
   STATUS[97].EXT.BIT29 := FALSE;
   STATUS[97].EXT.BIT30 := FALSE;
   STATUS[97].EXT.BIT31 := FALSE;
   STATUS[97].EXT.ModeBit1 := FALSE;
   STATUS[97].EXT.ModeBit2 := FALSE;
   STATUS[97].EXT.ModeBit3 := FALSE;
   STATUS[97].EXT.BIT19 := FALSE;
   STATUS[97].EXT.BIT20 := FALSE;
   STATUS[97].EXT.AlarmSuppressed := FALSE;
   STATUS[97].EXT.AlarmPrsent := FALSE;
   STATUS[97].EXT.AlarmFailUnAck := FALSE;
   STATUS[97].Status := 0;
   STATUS[97].TimeStamp := 16#0000;
   STATUS[98].VALUE := 0.0;
   STATUS[98].TRIGVALUE := 0.0;
   STATUS[98].EXT.AlarmWarnUnAck := FALSE;
   STATUS[98].EXT.AckRequired := FALSE;
   STATUS[98].EXT.Maintanence := FALSE;
   STATUS[98].EXT.Operation := FALSE;
   STATUS[98].EXT.Forced := FALSE;
   STATUS[98].EXT.BIT29 := FALSE;
   STATUS[98].EXT.BIT30 := FALSE;
   STATUS[98].EXT.BIT31 := FALSE;
   STATUS[98].EXT.ModeBit1 := FALSE;
   STATUS[98].EXT.ModeBit2 := FALSE;
   STATUS[98].EXT.ModeBit3 := FALSE;
   STATUS[98].EXT.BIT19 := FALSE;
   STATUS[98].EXT.BIT20 := FALSE;
   STATUS[98].EXT.AlarmSuppressed := FALSE;
   STATUS[98].EXT.AlarmPrsent := FALSE;
   STATUS[98].EXT.AlarmFailUnAck := FALSE;
   STATUS[98].Status := 0;
   STATUS[98].TimeStamp := 16#0000;
   STATUS[99].VALUE := 0.0;
   STATUS[99].TRIGVALUE := 0.0;
   STATUS[99].EXT.AlarmWarnUnAck := FALSE;
   STATUS[99].EXT.AckRequired := FALSE;
   STATUS[99].EXT.Maintanence := FALSE;
   STATUS[99].EXT.Operation := FALSE;
   STATUS[99].EXT.Forced := FALSE;
   STATUS[99].EXT.BIT29 := FALSE;
   STATUS[99].EXT.BIT30 := FALSE;
   STATUS[99].EXT.BIT31 := FALSE;
   STATUS[99].EXT.ModeBit1 := FALSE;
   STATUS[99].EXT.ModeBit2 := FALSE;
   STATUS[99].EXT.ModeBit3 := FALSE;
   STATUS[99].EXT.BIT19 := FALSE;
   STATUS[99].EXT.BIT20 := FALSE;
   STATUS[99].EXT.AlarmSuppressed := FALSE;
   STATUS[99].EXT.AlarmPrsent := FALSE;
   STATUS[99].EXT.AlarmFailUnAck := FALSE;
   STATUS[99].Status := 0;
   STATUS[99].TimeStamp := 16#0000;
   STATUS[100].VALUE := 0.0;
   STATUS[100].TRIGVALUE := 0.0;
   STATUS[100].EXT.AlarmWarnUnAck := FALSE;
   STATUS[100].EXT.AckRequired := FALSE;
   STATUS[100].EXT.Maintanence := FALSE;
   STATUS[100].EXT.Operation := FALSE;
   STATUS[100].EXT.Forced := FALSE;
   STATUS[100].EXT.BIT29 := FALSE;
   STATUS[100].EXT.BIT30 := FALSE;
   STATUS[100].EXT.BIT31 := FALSE;
   STATUS[100].EXT.ModeBit1 := FALSE;
   STATUS[100].EXT.ModeBit2 := FALSE;
   STATUS[100].EXT.ModeBit3 := FALSE;
   STATUS[100].EXT.BIT19 := FALSE;
   STATUS[100].EXT.BIT20 := FALSE;
   STATUS[100].EXT.AlarmSuppressed := FALSE;
   STATUS[100].EXT.AlarmPrsent := FALSE;
   STATUS[100].EXT.AlarmFailUnAck := FALSE;
   STATUS[100].Status := 0;
   STATUS[100].TimeStamp := 16#0000;
   STATUS[101].VALUE := 0.0;
   STATUS[101].TRIGVALUE := 0.0;
   STATUS[101].EXT.AlarmWarnUnAck := FALSE;
   STATUS[101].EXT.AckRequired := FALSE;
   STATUS[101].EXT.Maintanence := FALSE;
   STATUS[101].EXT.Operation := FALSE;
   STATUS[101].EXT.Forced := FALSE;
   STATUS[101].EXT.BIT29 := FALSE;
   STATUS[101].EXT.BIT30 := FALSE;
   STATUS[101].EXT.BIT31 := FALSE;
   STATUS[101].EXT.ModeBit1 := FALSE;
   STATUS[101].EXT.ModeBit2 := FALSE;
   STATUS[101].EXT.ModeBit3 := FALSE;
   STATUS[101].EXT.BIT19 := FALSE;
   STATUS[101].EXT.BIT20 := FALSE;
   STATUS[101].EXT.AlarmSuppressed := FALSE;
   STATUS[101].EXT.AlarmPrsent := FALSE;
   STATUS[101].EXT.AlarmFailUnAck := FALSE;
   STATUS[101].Status := 0;
   STATUS[101].TimeStamp := 16#0000;
   STATUS[102].VALUE := 0.0;
   STATUS[102].TRIGVALUE := 0.0;
   STATUS[102].EXT.AlarmWarnUnAck := FALSE;
   STATUS[102].EXT.AckRequired := FALSE;
   STATUS[102].EXT.Maintanence := FALSE;
   STATUS[102].EXT.Operation := FALSE;
   STATUS[102].EXT.Forced := FALSE;
   STATUS[102].EXT.BIT29 := FALSE;
   STATUS[102].EXT.BIT30 := FALSE;
   STATUS[102].EXT.BIT31 := FALSE;
   STATUS[102].EXT.ModeBit1 := FALSE;
   STATUS[102].EXT.ModeBit2 := FALSE;
   STATUS[102].EXT.ModeBit3 := FALSE;
   STATUS[102].EXT.BIT19 := FALSE;
   STATUS[102].EXT.BIT20 := FALSE;
   STATUS[102].EXT.AlarmSuppressed := FALSE;
   STATUS[102].EXT.AlarmPrsent := FALSE;
   STATUS[102].EXT.AlarmFailUnAck := FALSE;
   STATUS[102].Status := 0;
   STATUS[102].TimeStamp := 16#0000;
   STATUS[103].VALUE := 0.0;
   STATUS[103].TRIGVALUE := 0.0;
   STATUS[103].EXT.AlarmWarnUnAck := FALSE;
   STATUS[103].EXT.AckRequired := FALSE;
   STATUS[103].EXT.Maintanence := FALSE;
   STATUS[103].EXT.Operation := FALSE;
   STATUS[103].EXT.Forced := FALSE;
   STATUS[103].EXT.BIT29 := FALSE;
   STATUS[103].EXT.BIT30 := FALSE;
   STATUS[103].EXT.BIT31 := FALSE;
   STATUS[103].EXT.ModeBit1 := FALSE;
   STATUS[103].EXT.ModeBit2 := FALSE;
   STATUS[103].EXT.ModeBit3 := FALSE;
   STATUS[103].EXT.BIT19 := FALSE;
   STATUS[103].EXT.BIT20 := FALSE;
   STATUS[103].EXT.AlarmSuppressed := FALSE;
   STATUS[103].EXT.AlarmPrsent := FALSE;
   STATUS[103].EXT.AlarmFailUnAck := FALSE;
   STATUS[103].Status := 0;
   STATUS[103].TimeStamp := 16#0000;
   STATUS[104].VALUE := 0.0;
   STATUS[104].TRIGVALUE := 0.0;
   STATUS[104].EXT.AlarmWarnUnAck := FALSE;
   STATUS[104].EXT.AckRequired := FALSE;
   STATUS[104].EXT.Maintanence := FALSE;
   STATUS[104].EXT.Operation := FALSE;
   STATUS[104].EXT.Forced := FALSE;
   STATUS[104].EXT.BIT29 := FALSE;
   STATUS[104].EXT.BIT30 := FALSE;
   STATUS[104].EXT.BIT31 := FALSE;
   STATUS[104].EXT.ModeBit1 := FALSE;
   STATUS[104].EXT.ModeBit2 := FALSE;
   STATUS[104].EXT.ModeBit3 := FALSE;
   STATUS[104].EXT.BIT19 := FALSE;
   STATUS[104].EXT.BIT20 := FALSE;
   STATUS[104].EXT.AlarmSuppressed := FALSE;
   STATUS[104].EXT.AlarmPrsent := FALSE;
   STATUS[104].EXT.AlarmFailUnAck := FALSE;
   STATUS[104].Status := 0;
   STATUS[104].TimeStamp := 16#0000;
   STATUS[105].VALUE := 0.0;
   STATUS[105].TRIGVALUE := 0.0;
   STATUS[105].EXT.AlarmWarnUnAck := FALSE;
   STATUS[105].EXT.AckRequired := FALSE;
   STATUS[105].EXT.Maintanence := FALSE;
   STATUS[105].EXT.Operation := FALSE;
   STATUS[105].EXT.Forced := FALSE;
   STATUS[105].EXT.BIT29 := FALSE;
   STATUS[105].EXT.BIT30 := FALSE;
